        SP_HPivRnd_18_Xe.trans.X := g_H_sideplateDIST + NOZZLE_RADIUS;
        SP_HPivRnd_18_Xs.trans.X := g_H_sideplateDIST + NOZZLE_RADIUS + 50 ;
        SP_gPivRnd_18_Xe.trans.X := ( g_H_sideplateDIST + NOZZLE_RADIUS ) * (-1);
        SP_gPivRnd_18_Xs.trans.X := ( g_H_sideplateDIST + NOZZLE_RADIUS + 50) * (-1);

        SP_HPivRnd_18_Xe.trans.y := yy_SRCH_Target ;
        SP_HPivRnd_18_Xs.trans.y := yy_SRCH_Target;
        SP_gPivRnd_18_Xe.trans.y := yy_SRCH_Target ;
        SP_gPivRnd_18_Xs.trans.y := yy_SRCH_Target;

        SP_HPivRnd_18_Xe.trans.z := zz_SRCH_Target * (-1) ;
        SP_HPivRnd_18_Xs.trans.z := zz_SRCH_Target * (-1) ;
        SP_gPivRnd_18_Xe.trans.z := zz_SRCH_Target * (-1) ;
        SP_gPivRnd_18_Xs.trans.z := zz_SRCH_Target * (-1) ;

 !!!!!!!!!!!!!!!!!!!!!!!!!!!!!!!!!!!!!!!!!!!!!!!!!!!!!!!!!!!!!!!!!!!!!!!!!!!!!

        SP_hPivCam_18_Xe.trans.X := g_H_sideplateDIST - NOZZLE_RADIUS;
        SP_hPivCam_18_Xs.trans.X := g_H_sideplateDIST - NOZZLE_RADIUS - 50 ;
        SP_gPivCam_18_Xe.trans.X := (g_H_sideplateDIST -  NOZZLE_RADIUS) *(-1);
        SP_gPivCam_18_Xs.trans.X := (g_H_sideplateDIST - NOZZLE_RADIUS - 50) * (-1) ;

        SP_hPivCam_18_Xe.trans.y := yy_SRCH_Target ;
        SP_hPivCam_18_Xs.trans.y := yy_SRCH_Target;
        SP_gPivCam_18_Xe.trans.y := yy_SRCH_Target ;
        SP_gPivCam_18_Xs.trans.y := yy_SRCH_Target;

        SP_hPivCam_18_Xe.trans.z := zz_SRCH_Target * (-1) ;
        SP_hPivCam_18_Xs.trans.z := zz_SRCH_Target * (-1) ;
        SP_gPivCam_18_Xe.trans.z := zz_SRCH_Target * (-1) ;
        SP_gPivCam_18_Xs.trans.z := zz_SRCH_Target * (-1) ;

        SP_HPivRnd_PJ_Xe.trans.X := g_H_sideplateDIST - NOZZLE_RADIUS - SIDEPLATE;
        SP_HPivRnd_PJ_Xs.trans.X := g_H_sideplateDIST - NOZZLE_RADIUS - SIDEPLATE - 50;
        SP_gPivRnd_PJ_Xe.trans.X := (g_H_sideplateDIST - NOZZLE_RADIUS - SIDEPLATE) *(-1);
        SP_gPivRnd_PJ_Xs.trans.X := (g_H_sideplateDIST - NOZZLE_RADIUS - SIDEPLATE - 50) * (-1);

        SP_HPivRnd_PJ_Xe.trans.y := yy_SRCH_Target;
        SP_HPivRnd_PJ_Xs.trans.y := yy_SRCH_Target;
        SP_gPivRnd_PJ_Xe.trans.y := yy_SRCH_Target;
        SP_gPivRnd_PJ_Xs.trans.y := yy_SRCH_Target;

        SP_HPivRnd_PJ_Xe.trans.z := zz_SRCH_Target * (-1);
        SP_HPivRnd_PJ_Xs.trans.z := zz_SRCH_Target * (-1);
        SP_gPivRnd_PJ_Xe.trans.z := zz_SRCH_Target * (-1) ;
        SP_gPivRnd_PJ_Xs.trans.z := zz_SRCH_Target * (-1) ;

 !!!!!!!!!!!!!!!!!!!!!!!!!!!!!!!!!!!!!!!!!!!!!!!!!!!!!!!!!!!!!!!!!!!!!!!!!!!!!

        SP_hPivCam_PJ_Xe.trans.X := g_H_sideplateDIST + SIDEPLATE + NOZZLE_RADIUS;
        SP_hPivCam_PJ_Xs.trans.X := g_H_sideplateDIST + SIDEPLATE + NOZZLE_RADIUS + 50;
        SP_gPivCam_PJ_Xe.trans.X := (g_H_sideplateDIST + SIDEPLATE + NOZZLE_RADIUS) * (-1);
        SP_gPivCam_PJ_Xs.trans.X := (g_H_sideplateDIST + SIDEPLATE + NOZZLE_RADIUS + 50) * (-1);

        SP_hPivCam_PJ_Xe.trans.y := yy_SRCH_Target;
        SP_hPivCam_PJ_Xs.trans.y := yy_SRCH_Target;
        SP_gPivCam_PJ_Xe.trans.y := yy_SRCH_Target;
        SP_gPivCam_PJ_Xs.trans.y := yy_SRCH_Target;

        SP_hPivCam_PJ_Xe.trans.z := zz_SRCH_Target * (-1);
        SP_hPivCam_PJ_Xs.trans.z := zz_SRCH_Target * (-1);
        SP_gPivCam_PJ_Xe.trans.z := zz_SRCH_Target * (-1);
        SP_gPivCam_PJ_Xs.trans.z := zz_SRCH_Target * (-1);

!!!!!!!!!!!!!!!!!!!!!!!!!!!!!!!!!!!!!!!!!!!!!!!!!!!!!!!!!!!!!!!!!!!!!!!!!!!!!!!!!!!!!!!!!!!!!!!!!!!!!!
        SP_GRnd_Side_XE.TRANS.X := (g_H_sideplateDIST + NOZZLE_RADIUS) *(-1);
        SP_GRnd_Side_XS.TRANS.X := (g_H_sideplateDIST + NOZZLE_RADIUS + 50) *(-1);
        SP_GRnd_Side_XE.trans.y := yy_SRCH_Target;
        SP_GRnd_Side_XS.trans.y := yy_SRCH_Target;
        SP_GRnd_Side_XE.trans.z := zz_SRCH_Target * (-1);
        SP_GRnd_Side_XS.trans.z := zz_SRCH_Target * (-1);
        SP_GRnd_Side_XS.extax.eax_b := 0;
        SP_GRnd_Side_XS.extax.eax_c := 90;
        SP_GRnd_Side_XE.extax := SP_GRnd_Side_XS.extax;

        SP_HRnd_Side_XE.TRANS.X := (g_H_sideplateDIST + NOZZLE_RADIUS) ;
        SP_HRnd_Side_XS.TRANS.X := (g_H_sideplateDIST + NOZZLE_RADIUS + 50) ;
        SP_HRnd_Side_XE.trans.y := yy_SRCH_Target;
        SP_HRnd_Side_XS.trans.y := yy_SRCH_Target;
        SP_HRnd_Side_XE.trans.z := zz_SRCH_Target * (-1);
        SP_HRnd_Side_XS.trans.z := zz_SRCH_Target * (-1);
        SP_HRnd_Side_XS.extax.eax_b := 0;
        SP_HRnd_Side_XS.extax.eax_c := -90;
        SP_HRnd_Side_XE.extax := SP_HRnd_Side_XS.extax;

        SP_GCam_Side_XE.TRANS.X := (g_H_sideplateDIST + NOZZLE_RADIUS + SIDEPLATE) *(-1);
        SP_GCam_Side_XS.TRANS.X := (g_H_sideplateDIST + NOZZLE_RADIUS + SIDEPLATE + 50) *(-1);
        SP_GCam_Side_XE.trans.y := yy_SRCH_Target;
        SP_GCam_Side_XS.trans.y := yy_SRCH_Target;
        SP_GCam_Side_XE.trans.z := zz_SRCH_Target * (-1);
        SP_GCam_Side_XS.trans.z := zz_SRCH_Target * (-1);
        SP_GCam_Side_XE.extax := g29.extax;
        SP_GCam_Side_XS.extax := g29.extax;

        SP_HCam_Side_XE.TRANS.X := (g_H_sideplateDIST + NOZZLE_RADIUS + SIDEPLATE) ;
        SP_HCam_Side_XS.TRANS.X := (g_H_sideplateDIST + NOZZLE_RADIUS + SIDEPLATE + 50) ;
        SP_HCam_Side_XE.trans.y := yy_SRCH_Target;
        SP_HCam_Side_XS.trans.y := yy_SRCH_Target;
        SP_HCam_Side_XE.trans.z := zz_SRCH_Target * (-1);
        SP_HCam_Side_XS.trans.z := zz_SRCH_Target * (-1);
        SP_HCam_Side_XE.extax := H29.extax;
        SP_HCam_Side_XS.extax := H29.extax;

        SP_Piv0ut_GXe.trans.X := (g_H_sideplateDIST - NOZZLE_RADIUS) * (-1) ;
        SP_Piv0ut_GXs.trans.X := (g_H_sideplateDIST - NOZZLE_RADIUS - 50) * (-1) ;
        SP_Piv0ut_HXe.trans.X := (g_H_sideplateDIST - NOZZLE_RADIUS)  ;
        SP_Piv0ut_HXs.trans.X := (g_H_sideplateDIST - NOZZLE_RADIUS - 50)  ;

        SP_Piv0ut_GXe.trans.y := yy_SRCH_Target ;
        SP_Piv0ut_GXs.trans.y := yy_SRCH_Target ;
        SP_Piv0ut_GXe.trans.z := zz_SRCH_Target * (-1);
        SP_Piv0ut_GXs.trans.z := zz_SRCH_Target * (-1);

        SP_Piv0ut_HXe.trans.y := yy_SRCH_Target ;
        SP_Piv0ut_HXs.trans.y := yy_SRCH_Target ;
        SP_Piv0ut_HXe.trans.z := zz_SRCH_Target * (-1);
        SP_Piv0ut_HXs.trans.z := zz_SRCH_Target * (-1);

        IF pivCAM = TRUE THEN
            XH0E.TRANS.X := (g_H_sideplateDIST + SIDEPLATE + NOZZLE_RADIUS);
            XH19E.TRANS.X := (g_H_sideplateDIST + SIDEPLATE + NOZZLE_RADIUS);
            XH29E.TRANS.X := (g_H_sideplateDIST + SIDEPLATE + NOZZLE_RADIUS);

            XG0E.TRANS.X := (g_H_sideplateDIST + SIDEPLATE + NOZZLE_RADIUS) * (-1);
            XG19E.TRANS.X := (g_H_sideplateDIST + SIDEPLATE + NOZZLE_RADIUS) * (-1);
            XG29E.TRANS.X :=  (g_H_sideplateDIST + SIDEPLATE + NOZZLE_RADIUS) * (-1);

            XL49E.TRANS.X := (g_H_sideplateDIST + SIDEPLATE + NOZZLE_RADIUS);
            XM49E.TRANS.X := (g_H_sideplateDIST - NOZZLE_RADIUS) * (-1) ;
        ELSEIF PIVCAM = FALSE THEN
            XH0E.TRANS.X := (g_H_sideplateDIST + NOZZLE_RADIUS);
            XH19E.TRANS.X := (g_H_sideplateDIST  + NOZZLE_RADIUS);
            XH29E.TRANS.X := (g_H_sideplateDIST  + NOZZLE_RADIUS);

            XG0E.TRANS.X := (g_H_sideplateDIST + NOZZLE_RADIUS) * (-1);
            XG19E.TRANS.X := (g_H_sideplateDIST + NOZZLE_RADIUS) * (-1);
            XG29E.TRANS.X :=  (g_H_sideplateDIST + NOZZLE_RADIUS) * (-1);

            XL49E.TRANS.X := (g_H_sideplateDIST  + NOZZLE_RADIUS);
            XM49E.TRANS.X := (g_H_sideplateDIST - SIDEPLATE - NOZZLE_RADIUS) * (-1) ;
        ENDIF
        WAITTIME\INPOS,.2;
    ENDPROC

    PROC Piv_side_Welds(string RND_OR_NOT)

	 IF PIVOT_USED = 6089330 OR PIVOT_USED = 6802774 OR PIVOT_USED = 6870131 OR PIVOT_USED = 6845931 THEN
     !!  THIS IS FOR A 42H, 33H AND 24H
	    pivCAM := FALSE;

 	ELSEIF PIVOT_USED =  674961 OR PIVOT_USED = 350404 OR PIVOT_USED = 6099018 THEN
     !!  THIS IS FOR 77F THRU 120F AND 18H !
        pivCAM := TRUE;

	ELSE STOP;

	ENDIF

	WAITTIME\INPOS,.1;

	IF RND_OR_NOT = "G" AND pivCAM = TRUE THEN
		GOTO G_CAM_SIDE_WELDS;

	ELSEIF RND_OR_NOT = "G" AND pivCAM = FALSE THEN
		GOTO G_RND_SIDE_WELDS;

	ELSEIF RND_OR_NOT = "H" AND pivCAM = TRUE THEN
		GOTO H_CAM_SIDE_WELDS;

	ELSEIF RND_OR_NOT = "H" AND pivCAM = FALSE THEN
		GOTO H_RND_SIDE_WELDS;

    ELSE STOP;

	ENDIF
 G_RND_SIDE_WELDS:
        ! This is executed only if the Pivot is ROUND in Shape
       	ActUnit STN1;
        BEGIN_TEST_WELD_Grnd_OUTSIDE:
        MoveJ Offs(SP_GRnd_Side_XS, -300, 0, 0), V500, z10, tWeldGun\WObj:=wobj_PivCam;
        MoveL Offs(SP_GRnd_Side_XS, -50, 0, 0), V500, z5, tWeldGun\WObj:=wobj_PivCam;
        Search_1D SR_GSide_X\SearchStop:=gX_SideFOUND, SP_GRnd_Side_XS, SP_GRnd_Side_XE, v50, tWeldGun\WObj:=wobj_PivCam\SchSpeed:=10;
        MoveL Offs(SP_GRnd_Side_XS, -100, 0, 0), V500, z5, tWeldGun\WObj:=wobj_PivCam;
        MoveJ Offs(SP_GRnd_Side_YS, -120, 100, 0), V500, z10, tWeldGun\WObj:=wobjHsideplate;
        PivG_SideYZ_XSET_18_R1 gX_SideFOUND ;
        MoveL offs(SP_GRnd_Side_YS,-120,75,0), V500, z5, tWeldGun\WObj:=wobjHsideplate;
        MoveL offs(SP_GRnd_Side_YS,0,75,0), V500, z5, tWeldGun\WObj:=wobjHsideplate;
        Search_1D SR_GSide_Y\SearchStop:=gY_SideFOUND, SP_GRnd_Side_YS, SP_GRnd_Side_YE, v300, tWeldGun\WObj:=wobjHsideplate\SchSpeed:=10;
  		MoveL gY_SideFOUND, V500, z1, tWeldGun\WObj:=wobjHsideplate;
        WaitTime\InPos, 1;
        PivFOUND_Y := CRobT(\Tool:=tWeldgun\WObj:=obSTN1);
        WaitTime\InPos, 1;
        MoveL offs(SP_GRnd_Side_YS,0,50,0), V500, z5, tWeldGun\WObj:=wobjHsideplate;
        MoveL offs(SP_GRnd_Side_YS,-150,100,0), V500, z10, tWeldGun\WObj:=wobjHsideplate;
        MoveJ offs(SP_GRnd_Side_ZS,-150,0,100), V500, z10, tWeldGun\WObj:=wobjHsideplate;
        MoveL offs(SP_GRnd_Side_ZS,0,0,50), v400, z10, tWeldGun\WObj:=wobjHsideplate;
        Search_1D SR_GSide_Z\SearchStop:=gZ_SideFOUND, SP_GRnd_Side_ZS, SP_GRnd_Side_ZE, v300, tWeldGun\WObj:=wobjHsideplate\SchSpeed:=10;
  		MoveL gZ_SideFOUND, V500, z1, tWeldGun\WObj:=wobjHsideplate;
        WaitTime\InPos, 1;
        PivFOUND_Z := CRobT(\Tool:=tWeldgun\WObj:=obSTN1);
        WaitTime\InPos, 1;
        MoveL offs(SP_GRnd_Side_ZS,0,0,75), V500, z5, tWeldGun\WObj:=wobjHsideplate;
        PivWobj_Translation_Locator wobj_PivCam, PivFOUND_Y, PivFOUND_Z, WPIVOTANGLE;
        WaitTime\inpos, 1;
        MoveJ offs(SP_GRnd_Side_ZS,-300,0,75), V500, z10, tWeldGun\WObj:=wobjHsideplate;
        MoveJ Offs(GRnd_SidePIV_S,-300,200,0), V500, z10, tWeldGun\WObj:=wobj_PivCam;
        Search_1D SRpivotYhelperGsideRound,Offs(SPpivotYhelperGsideRoundE,0,30,0), SPpivotYhelperGsideRoundE, v100, tWeldGun\WObj:=wobj_PivCam\SchSpeed:=10;
        MoveJ Offs(GRnd_SidePIV_S,-300,200,0), V500, z10, tWeldGun\WObj:=wobj_PivCam;
        MoveJ offs(GRnd_SidePIV_S,-300,0,0), V500, z10, tWeldGun\WObj:=wobj_PivCam;
        PDispSet SRpivotYhelperGsideRound;
        ArcLStart GRnd_SidePIV_S, v100, smGH40A, wdGH40B\Weave:=wvGH40B, z1, tWeldGun\WObj:=wobj_PivCam;
		ArcL Offs(GRnd_SidePIV_S,0,0,5), v100, smGH40A, wdGH40B\Weave:=wvGH40B, z1, tWeldGun\WObj:=wobj_PivCam;
		WaitTime\InPos, 0.5;
		ArcL GRnd_SidePIV_Sm, v100, smGH40A, wdGH40B\Weave:=wvGH40B, z1, tWeldGun\WObj:=wobj_PivCam;
		ArcL GRnd_SidePIV_M, v100, smGH40A, wdGH40A\Weave:=wvGH40A, z1, tWeldGun\WObj:=wobj_PivCam;
		ArcL GRnd_SidePIV_Em, v100, smGH40A, wdGH40C\Weave:=wv0, z1, tWeldGun\WObj:=wobj_PivCam;
		ArcLEnd GRnd_SidePIV_E, v100, smGH40A, wdGH40C\Weave:=wv0, z1, tWeldGun\WObj:=wobj_PivCam;
        PDispOff;
        MoveL offs(GRnd_SidePIV_E,-50,0,0), V500, z10, tWeldGun\WObj:=wobj_PivCam;
        MoveJ offs(GRnd_SidePIV_E,-600,0,0), V500, z10, tWeldGun\WObj:=wobj_PivCam;
        WELDED_GRND_OUTSIDE:
        GOTO GLUED_THE_PIV_SIDES;
G_CAM_SIDE_WELDS:
        ! This is executed only if the Pivot is CAM in Shape
       	ActUnit STN1;
        BEGIN_TEST_WELD_GCam_OUTSIDE:
        PivG_SideYZ_XSET_18_R1 Gx_weld_piv;
        WAITTIME\INPOS, 1;
        firstYthentheZ:
        MoveJ Offs(SP_GCam_Side_YS, -175, 100, 0), V500, z10, tWeldGun\WObj:=wobjHsideplate;
        MoveL offs(SP_GCam_Side_YS,0,75,0), V500, z5, tWeldGun\WObj:=wobjHsideplate;
        Search_1D SR_GSide_Y\SearchStop:=gY_SideFOUND, SP_GCam_Side_YS, SP_GCam_Side_YE, v300, tWeldGun\WObj:=wobjHsideplate\SchSpeed:=10;
  		MoveL gY_SideFOUND, V500, z1, tWeldGun\WObj:=wobjHsideplate;
        WaitTime\InPos, 1;
        PivFOUND_Y := CRobT(\Tool:=tWeldgun\WObj:=obSTN1);
        WaitTime\InPos, 1;
        MoveL offs(SP_GCam_Side_YS,0,50,0), V500, z5, tWeldGun\WObj:=wobjHsideplate;
        MoveL offs(SP_GCam_Side_YS,-150,100,0), V500, z10, tWeldGun\WObj:=wobjHsideplate;
        nowtheZ:
        MoveJ offs(SP_GCam_Side_ZS,-150,0,100), V500, z10, tWeldGun\WObj:=wobjHsideplate;
        MoveL offs(SP_GCam_Side_ZS,0,0,50), v400, z10, tWeldGun\WObj:=wobjHsideplate;
        Search_1D SR_GSide_Z\SearchStop:=gZ_SideFOUND, SP_GCam_Side_ZS, SP_GCam_Side_ZE, v300, tWeldGun\WObj:=wobjHsideplate\SchSpeed:=10;
  		MoveL gZ_SideFOUND, V500, z1, tWeldGun\WObj:=wobjHsideplate;
        WaitTime\InPos, 1;
        PivFOUND_Z := CRobT(\Tool:=tWeldgun\WObj:=obSTN1);
        WaitTime\InPos, 1;
        MoveL offs(SP_GCam_Side_ZS,0,0,75), V500, z5, tWeldGun\WObj:=wobjHsideplate;
        PivWobj_Translation_Locator wobj_PivCam, PivFOUND_Y, PivFOUND_Z, WPIVOTANGLE;
        WaitTime\inpos, 1;
        MoveL offs(SP_GCam_Side_ZS,-300,0,75), V500, z10, tWeldGun\WObj:=wobjHsideplate;
        MoveJ RelTooL(GCam_SidePIV_S,0,0,-350), V500, z10, tWeldGun\WObj:=wobj_PivCam;
        WELDED_GCAM_OUTSIDE:
        GOTO GLUED_THE_PIV_SIDES;
 H_CAM_SIDE_WELDS:
            ! This is executed only if the Pivot is CAM in Shape
       	ActUnit STN1;
        BEGIN_TEST_WELD_HCam_OUTSIDE:
        PivH_SideYZ_XSET_18_R1 hx_weld_piv;
        MoveJ Offs(SP_HCam_Side_YS, 200, 100, 0), V500, z10, tWeldGun\WObj:=wobjHsideplate;
        MoveL offs(SP_HCam_Side_YS,0,75,0), V500, z5, tWeldGun\WObj:=wobjHsideplate;
        Search_1D SR_HSide_Y\SearchStop:=hY_SideFOUND, SP_HCam_Side_YS, SP_HCam_Side_YE, v300, tWeldGun\WObj:=wobjHsideplate\SchSpeed:=10;
  		MoveL hY_SideFOUND, V500, z1, tWeldGun\WObj:=wobjHsideplate;
        WaitTime\InPos, 1;
        PivFOUND_Y := CRobT(\Tool:=tWeldgun\WObj:=obSTN1);
        WaitTime\InPos, 1;
        MoveL offs(SP_HCam_Side_YS,0,50,0), V500, z5, tWeldGun\WObj:=wobjHsideplate;
        MoveL offs(SP_HCam_Side_YS,150,100,0), V500, z10, tWeldGun\WObj:=wobjHsideplate;
        MoveJ offs(SP_HCam_Side_ZS,150,0,100), V500, z10, tWeldGun\WObj:=wobjHsideplate;
        MoveL offs(SP_HCam_Side_ZS,0,0,50), v400, z10, tWeldGun\WObj:=wobjHsideplate;
        Search_1D SR_HSide_Z\SearchStop:=hZ_SideFOUND, SP_HCam_Side_ZS, SP_HCam_Side_ZE, v300, tWeldGun\WObj:=wobjHsideplate\SchSpeed:=10;
  		MoveL hZ_SideFOUND, V500, z1, tWeldGun\WObj:=wobjHsideplate;
        WaitTime\InPos, 1;
        PivFOUND_Z := CRobT(\Tool:=tWeldgun\WObj:=obSTN1);
        WaitTime\InPos, 1;
        MoveL offs(SP_HCam_Side_ZS,0,0,75), V500, z5, tWeldGun\WObj:=wobjHsideplate;
        PivWobj_Translation_Locator wobj_PivCam, PivFOUND_Y, PivFOUND_Z, WPIVOTANGLE;
        WaitTime\inpos, 1;
        MoveL offs(SP_HCam_Side_ZS,0,-300,0), V500, z10, tWeldGun\WObj:=wobjHsideplate;
        MoveJ reltool(HCam_SidePIV_S,0,0,-300), V500, z10, tWeldGun\WObj:=wobj_PivCam;
        WELDED_HCAM_OUTSIDE:
        GOTO GLUED_THE_PIV_SIDES;
 H_RND_SIDE_WELDS:
        ! This is executed only if the Pivot is ROUND in Shape
       	ActUnit STN1;
        BEGIN_TEST_WELD_HRnd_OUTSIDE:
        MoveJ Offs(SP_HRnd_Side_XS, 300, 0, 0), V500, z10, tWeldGun\WObj:=wobj_PivCam;
        MoveL Offs(SP_HRnd_Side_XS, 50, 0, 0), V500, z5, tWeldGun\WObj:=wobj_PivCam;
        Search_1D SR_HSide_X\SearchStop:=hX_SideFOUND, SP_HRnd_Side_XS, SP_HRnd_Side_XE, v50, tWeldGun\WObj:=wobj_PivCam\SchSpeed:=10;
        MoveL Offs(SP_HRnd_Side_XS, 100, 0, 0), V500, z5, tWeldGun\WObj:=wobj_PivCam;
        PivH_SideYZ_XSET_18_R1 hX_SideFOUND;
        MoveJ Offs(SP_HRnd_Side_YS, 100, 100, 0), V500, z10, tWeldGun\WObj:=wobjHsideplate;
        MoveL offs(SP_HRnd_Side_YS,0,75,0), V500, z5, tWeldGun\WObj:=wobjHsideplate;
        Search_1D SR_HSide_Y\SearchStop:=hY_SideFOUND, SP_HRnd_Side_YS, SP_HRnd_Side_YE, v300, tWeldGun\WObj:=wobjHsideplate\SchSpeed:=10;
  		MoveL hY_SideFOUND, V500, z1, tWeldGun\WObj:=wobjHsideplate;
        WaitTime\InPos, 1;
        PivFOUND_Y := CRobT(\Tool:=tWeldgun\WObj:=obSTN1);
        WaitTime\InPos, 1;
        MoveL offs(SP_HRnd_Side_YS,0,50,0), V500, z5, tWeldGun\WObj:=wobjHsideplate;
        MoveL offs(SP_HRnd_Side_YS,150,100,0), V500, z10, tWeldGun\WObj:=wobjHsideplate;
        MoveJ offs(SP_HRnd_Side_ZS,150,0,100), V500, z10, tWeldGun\WObj:=wobjHsideplate;
        MoveL offs(SP_HRnd_Side_ZS,0,0,50), v400, z10, tWeldGun\WObj:=wobjHsideplate;
        Search_1D SR_HSide_Z\SearchStop:=hZ_SideFOUND, SP_HRnd_Side_ZS, SP_HRnd_Side_ZE, v300, tWeldGun\WObj:=wobjHsideplate\SchSpeed:=10;
  		MoveL hZ_SideFOUND, V500, z1, tWeldGun\WObj:=wobjHsideplate;
        WaitTime\InPos, 1;
        PivFOUND_Z := CRobT(\Tool:=tWeldgun\WObj:=obSTN1);
        WaitTime\InPos, 1;
        MoveL offs(SP_HRnd_Side_ZS,0,0,75), V500, z5, tWeldGun\WObj:=wobjHsideplate;
        PivWobj_Translation_Locator wobj_PivCam, PivFOUND_Y, PivFOUND_Z, WPIVOTANGLE;
        WaitTime\inpos, 1;
        MoveL offs(SP_HRnd_Side_ZS,300,0,75), V500, z10, tWeldGun\WObj:=wobjHsideplate;
        MoveJ Offs(HRnd_SidePIV_S,300,200,0), V500, z10, tWeldGun\WObj:=wobj_PivCam;
        Search_1D SRpivotYhelperHsideRound,Offs(SPpivotYhelperHsideRoundE,0,30,0), SPpivotYhelperHsideRoundE, v100, tWeldGun\WObj:=wobj_PivCam\SchSpeed:=10;
        MoveJ Offs(HRnd_SidePIV_S,300,200,0), V500, z10, tWeldGun\WObj:=wobj_PivCam;
        MoveJ offs(HRnd_SidePIV_S,300,0,0), V500, z10, tWeldGun\WObj:=wobj_PivCam;
        MoveJ offs(HRnd_SidePIV_S,300,0,0), V500, z10, tWeldGun\WObj:=wobj_PivCam;
        PDispSet SRpivotYhelperHsideRound;
 		ArcLStart HRnd_SidePIV_S, v100, smGH40A, wdGH40B\Weave:=wvGH40B, z1, tWeldGun\WObj:=wobj_PivCam;
		ArcL Offs(HRnd_SidePIV_S,0,0,5), v100, smGH40A, wdGH40B\Weave:=wvGH40B, z1, tWeldGun\WObj:=wobj_PivCam;
		WaitTime\InPos, 0.5;
		ArcL HRnd_SidePIV_Sm, v100, smGH40A, wdGH40B\Weave:=wvGH40B, z1, tWeldGun\WObj:=wobj_PivCam;
		ArcL HRnd_SidePIV_M, v100, smGH40A, wdGH40A\Weave:=wvGH40A, z1, tWeldGun\WObj:=wobj_PivCam;
		ArcL HRnd_SidePIV_Em, v100, smGH40A, wdGH40C\Weave:=wv0, z1, tWeldGun\WObj:=wobj_PivCam;
		ArcLEnd HRnd_SidePIV_E, v100, smGH40A, wdGH40C\Weave:=wv0, z1, tWeldGun\WObj:=wobj_PivCam;
        PDispOff;
        MoveL offs(HRnd_SidePIV_E,50,0,0), V500, z10, tWeldGun\WObj:=wobj_PivCam;
        MoveJ offs(HRnd_SidePIV_E,600,0,0), V500, z10, tWeldGun\WObj:=wobj_PivCam;
        WELDED_HRnd_OUTSIDE:
        GOTO GLUED_THE_PIV_SIDES;
      GLUED_THE_PIV_SIDES:
    ENDPROC

        PROC Piv0ut2Fwrap_X18_R1()

                SP_Piv0ut_Ye.trans.X := (hX_FOUND.TRANS.X) + (NOZZLE_RADIUS * 1.5)  ;
                SP_Piv0ut_Ys.trans.X := (hX_FOUND.TRANS.X) + (NOZZLE_RADIUS * 1.5)  ;
                SP_Piv0ut_Ye.trans.y := NOZZLE_RADIUS ;
                SP_Piv0ut_Ys.trans.y := NOZZLE_RADIUS + 55;

                SP_Piv0ut_Ye.trans.z := wobjHpivot.oframe.trans.Z - 164 ;
                SP_Piv0ut_Ys.trans.z := wobjHpivot.oframe.trans.Z - 164 ;
                SP_Piv0ut_Ze.trans.X := (hX_FOUND.TRANS.X) + (NOZZLE_RADIUS*1.5) ;
                SP_Piv0ut_Zs.trans.X := (hX_FOUND.TRANS.X) + (NOZZLE_RADIUS*1.5) ;

                SP_Piv0ut_Ze.trans.Y := 36;
                SP_Piv0ut_Zs.trans.Y := 36;
                SP_Piv0ut_Ze.trans.z := (wobjHpivot.oframe.trans.Z)  - hfixconst + nozzle_radius ;
                SP_Piv0ut_Zs.trans.z := (wobjHpivot.oframe.trans.Z - HFIXCONST + NOZZLE_RADIUS + 50) ;
            over_it:
    ENDPROC

    PROC Weld_Piv0ut_2FWrap()
       ActUnit STN1;
       PDispOff;
       PDispOff;
       MoveJ pjthomeSTA1zero, vCellSpeed, fine, tWeldGun\WObj:=wobj0;
       MoveJ RelTool(SP_Piv0ut_GXs,0,0,-650), V500, z20, tWeldGun\WObj:=wobj_PivCam;
       MoveL RelTool(SP_Piv0ut_GXs,0,0,-150), V500, z5, tWeldGun\WObj:=wobj_PivCam;
       PDispOff;
       MoveL SP_Piv0ut_GXs, V500, z1, tWeldGun\WObj:=wobj_PivCam;
       Search_1D SR_Gx\SearchStop:=gX_FOUND, SP_Piv0ut_GXs, SP_Piv0ut_GXe, v300, tWeldGun\WObj:=wobj_PivCam\SchSpeed:=10;
       MoveL RelTool(SP_Piv0ut_GXs,0,0,-50), V500, z5, tWeldGun\WObj:=wobj_PivCam;
       MoveL RelTool(SP_Piv0ut_HXs,0,0,-50), V500, z5, tWeldGun\WObj:=wobj_PivCam;
       Search_1D SR_Hx\SearchStop:=hX_FOUND, SP_Piv0ut_HXs, SP_Piv0ut_HXe, v300, tWeldGun\WObj:=wobj_PivCam\SchSpeed:=10;
       MoveL RelTool(SP_Piv0ut_HXs,0,0,-150), V500, z5, tWeldGun\WObj:=wobj_PivCam;
       Piv0ut2Fwrap_X18_R1;
       MoveJ Offs(SP_Piv0ut_Zs,0,-250,0), V500, z5, tWeldGun\WObj:=wobjHsideplate;
       MoveJ Offs(SP_Piv0ut_Zs,250,-250,0), V500, z5, tWeldGun\WObj:=wobjHsideplate;
       MoveJ Offs(SP_Piv0ut_Ys,250,0,50), V500, z5, tWeldGun\WObj:=wobjHsideplate;
       Search_1D SR_Piv_Y\SearchStop:=PivFOUND_Y, SP_Piv0ut_Ys, SP_Piv0ut_Ye, v300, tWeldGun\WObj:=wobjHsideplate\PrePDisp:=SR_Hx\SchSpeed:=10;
  	   MoveL PivFOUND_Y, V500, z1, tWeldGun\WObj:=wobjHsideplate;
       PDispOff;
       WaitTime\InPos, 1;
       PivFOUND_Y := CRobT(\Tool:=tWeldGun\WObj:=obSTN1);
       WaitTime\InPos, 1;
       MoveL Offs(SP_Piv0ut_Ys,0,50,0), V500, z5, tWeldGun\WObj:=wobjHsideplate;
       MoveL OFFS(SP_Piv0ut_Ys,250,0,50), V500, z5, tWeldGun\WObj:=wobjHsideplate;
       MoveJ OFFS(SP_Piv0ut_Zs,200,0,150), V500, z5, tWeldGun\WObj:=wobjHsideplate;
       MoveL OFFS(SP_Piv0ut_Zs,200,0,50), V500, z5, tWeldGun\WObj:=wobjHsideplate;
       Search_1D SR_Piv_Z\SearchStop:=PivFOUND_z, SP_Piv0ut_Zs, SP_Piv0ut_Ze, v300, tWeldGun\WObj:=wobjHsideplate\PrePDisp:=SR_Piv_Y\SchSpeed:=10;
  	   MoveL PivFOUND_z, V500, z1, tWeldGun\WObj:=wobjHsideplate;
       PDispOff;
       WaitTime\InPos, 1;
       PivFOUND_z := CRobT(\Tool:=tWeldGun\WObj:=obSTN1);
       WaitTime\InPos, 1;
       MoveL OFFS(SP_Piv0ut_Zs,0,-50,100), V500, z5, tWeldGun\WObj:=wobjHsideplate;
       MoveL OFFS(SP_Piv0ut_Zs,200,50,0), V500, z5, tWeldGun\WObj:=wobjHsideplate;
        PivWobj_Translation_Locator wobj_PivCam, PivFOUND_Y, PivFOUND_Z, WPIVOTANGLE;
        WaitTime\InPos, 1;
       !MoveL OFFS(SP_Piv0ut_Ys,200,-300,0), V500, z5, tWeldGun\WObj:=wobjHsideplate;
       MoveJ OFFS(SP_Piv0ut_Zs,200,-300,0), V500, z5, tWeldGun\WObj:=wobjHsideplate;
       MoveJ OFFS(SP_Piv0ut_Zs,-100,-300,0), V500, z5, tWeldGun\WObj:=wobjHsideplate;
       MoveJ OFFS(OSPiv2Fwrap_G1,100,-200,0), V500, z5, tWeldGun\WObj:=wobj_PivCam;
       !Y and Z SEARCH FOR DISP...03-19-18
       Search_1D SR_YPIVadj,Offs(SP_YPIVadj_e,0,-30,0), SP_YPIVadj_e, v300, tWeldGun\WObj:=wobj_PivCam\SchSpeed:=10;
       MoveJ OFFS(OSPiv2Fwrap_G1,100,-200,0), V500, z5, tWeldGun\WObj:=wobj_PivCam;
       Search_1D\Wire, SR_ZPIVadj, Offs(SP_ZPIVadj_e,0,-10,-30), SP_ZPIVadj_e, v300, tWeldGun\WObj:=wobj_PivCam\SchSpeed:=10;
       MoveJ OFFS(OSPiv2Fwrap_G1,100,-200,0), V500, z5, tWeldGun\WObj:=wobj_PivCam;
		SR_Gx.trans.y := SR_YPIVadj.trans.y;
		SR_Gx.trans.z := SR_ZPIVadj.trans.z;
		SR_Hx.trans.y := SR_YPIVadj.trans.y;
		SR_Hx.trans.z := SR_ZPIVadj.trans.z;
        WaitTime\InPos, 1;
        TPErase;
        TPErase;
       PDispSet SR_Gx;
	   ArcLStart OSPiv2Fwrap_G3, v100, smJKnofill, wdJKroot\Weave:=wvJKroot, z1, tWeldGun\WObj:=wobj_PivCam;
       PDispSet SR_Hx;
       ArcLEnd OSPiv2Fwrap_H3, v100, smJKnofill, wdJKroot\Weave:=wvJKroot, z1, tWeldGun\WObj:=wobj_PivCam;
       MoveL Offs(OSPiv2Fwrap_H3,0,-35,0), v100, z1, tWeldGun\WObj:=wobj_PivCam;
       PDispOff;
	   MoveL Offs(OSPiv2Fwrap_G1,35,-35,0), v300, z1, tWeldGun\WObj:=wobj_PivCam;
       PDispSet SR_Gx;
       ArcLStart OSPiv2Fwrap_G1, v100, smJK1, wdJK1\Weave:=wv0, z1, tWeldGun\WObj:=wobj_PivCam\Track:=track0;
	   ArcL OSPiv2Fwrap_G2, v100, smJK, wdJK1\Weave:=wv0, z1, tWeldGun\WObj:=wobj_PivCam\Track:=track0;
	   ArcL OSPiv2Fwrap_G3, v100, smJK, wdJK1\Weave:=wvJK, z1, tWeldGun\WObj:=wobj_PivCam\Track:=track0;
	   ArcLEnd OSPiv2Fwrap_G4, v100, smJKnofill, wdJK\Weave:=wvJK, z1, tWeldGun\WObj:=wobj_PivCam\Track:=trLM10hiteonly;
	   PDispOff;
       MoveL Offs(OSPiv2Fwrap_G4,0,-35,0), v100, z1, tWeldGun\WObj:=wobj_PivCam;
	   MoveL Offs(OSPiv2Fwrap_H1,-35,-35,0), v100, z1, tWeldGun\WObj:=wobj_PivCam;
       PDispSet SR_Hx;
       ArcLStart OSPiv2Fwrap_H1, v100, smJK1, wdJK1\Weave:=wv0, z1, tWeldGun\WObj:=wobj_PivCam\Track:=track0;
	   ArcL OSPiv2Fwrap_H2, v100, smJK, wdJK1\Weave:=wv0, z1, tWeldGun\WObj:=wobj_PivCam\Track:=track0;
	   ArcL OSPiv2Fwrap_H3, v100, smJK, wdJK1\Weave:=wvJK, z1, tWeldGun\WObj:=wobj_PivCam\Track:=track0;
	   !ArcL OSPiv2Fwrap_H4, v100, smJK, wdJK1\Weave:=wvJK, z1, tWeldGun\WObj:=wobj_PivCam\Track:=track0;
	   ArcLEnd Offs(OSPiv2Fwrap_H4,-10,0,0), v100, smJK, wdJK\Weave:=wvJK, z1, tWeldGun\WObj:=wobj_PivCam\Track:=trLM10hiteonly;
	   PDispOff;
       MoveL RelTool(OSPiv2Fwrap_H4,0,0,-100), V500, z5, tWeldGun\WObj:=wobj_PivCam;
       MoveL RelTool(OSPiv2Fwrap_H4,0,0,-600), V500, z5, tWeldGun\WObj:=wobj_PivCam;
       MoveL Offs(OSPiv2Fwrap_H4,0,-600,-800), V500, z5, tWeldGun\WObj:=wobj_PivCam;
	   MoveJ pjthomeSTA1zero, vCellSpeed, fine, tWeldGun\WObj:=wobj0;
       HIJKLMNOP:
    ENDPROC

!!!!!!!!!!!!!!!!!!!!!!!!!!!!!!!!!!!!!!!!!!!!!!!!!!!!
!!!!!!!!!!!!!!!!!!!!!!!!!!!!!!!!!!!!!!!!!!!!!!!!!!!!
    PROC SET_ANCHOR_SRCH()
    !!!!!!!!!!!THIS PROC HAS BEEN partially modified (6099135,6802707,6862141,6089394, 6850291,689234) these numbers MODIFIED FOR SEARCHING ANCHORS TOTALLY WITH THE NOZZLE 02-05-18!!!!!!!
!!!!!!!!!!!!!!!!REVISED 03-16-18 to add anchor_back X searches!!!!!
IF ANCHOR_USED = 689234 THEN
	! ANCHOR "Y BACK" SEARCH  L & R
	SP_AGBY_E.trans.x := (FAMILY_GX.trans.x + NOZZLE_RADIUS + SIDEPLATE + 107 ); ! 44 Represents the middle between the sideplate and anchor lug
	SP_AGBY_E.trans.y := -13.5;	!(yeager changed it 12-02-17)
	SP_AGBY_E.trans.z := -48.5; !(yeager changed it 12-02-17)

	SP_AGBY_S.trans.x := (FAMILY_GX.trans.x + NOZZLE_RADIUS + SIDEPLATE + 107 );
	SP_AGBY_S.trans.y := -53.5; !(yeager changed it 12-02-17)
	SP_AGBY_S.trans.z := -48.5; !(yeager changed it 12-02-17)

	SP_AHBY_E.trans.x := (FAMILY_HX.trans.x - NOZZLE_RADIUS - SIDEPLATE - 107 ); ! 44 Represents the middle between the sideplate and anchor lug
	SP_AHBY_E.trans.y := -13.5; !(yeager changed it 12-02-17)
	SP_AHBY_E.trans.z := -48.5; !(yeager changed it 12-02-17)

	SP_AHBY_S.trans.x := (FAMILY_HX.trans.x - NOZZLE_RADIUS - SIDEPLATE - 107 );
	SP_AHBY_S.trans.y := -53.5; !(yeager changed it 12-02-17)
	SP_AHBY_S.trans.z := -48.5;	!(yeager changed it 12-02-17)

IF WOTOX < 1300 THEN


  	! ANCHOR "Y FRONT" SEARCH  L & R (short)
	SP_AGFY_E.trans.x := (FAMILY_GX.trans.x + NOZZLE_RADIUS + SIDEPLATE + 56.75 ); !yeager changed it 12-04-17...was 106.75
	SP_AGFY_E.trans.y := 13.5;	!(yeager changed it 12-02-17)
	SP_AGFY_E.trans.z := 9;	!(yeager changed it 12-02-17)

	SP_AGFY_S.trans.x := (FAMILY_GX.trans.x + NOZZLE_RADIUS + SIDEPLATE + 56.75 ); !yeager changed it 12-04-17...was 106.75
	SP_AGFY_S.trans.y := 53.5;	!(yeager changed it 12-02-17)
	SP_AGFY_S.trans.z := 9;	!(yeager changed it 12-02-17)

	SP_AHFY_E.trans.x := (FAMILY_HX.trans.x - NOZZLE_RADIUS - SIDEPLATE - 56.75 ); !yeager changed it 12-04-17...was 106.75
	SP_AHFY_E.trans.y := 13.5;	!(yeager changed it 12-02-17)
	SP_AHFY_E.trans.z := 9;	!(yeager changed it 12-02-17)

	SP_AHFY_S.trans.x := (FAMILY_HX.trans.x - NOZZLE_RADIUS - SIDEPLATE - 56.75 ); !yeager changed it 12-04-17...was 106.75
	SP_AHFY_S.trans.y := 53.5;	!(yeager changed it 12-02-17)
	SP_AHFY_S.trans.z := 9;	!(yeager changed it 12-02-17)

ELSE

  	! ANCHOR "Y FRONT" SEARCH  L & R (long)
	SP_AGFY_E.trans.x := (FAMILY_GX.trans.x + NOZZLE_RADIUS + SIDEPLATE + 106.75 ); !yeager changed it 12-04-17...was 106.75
	SP_AGFY_E.trans.y := 13.5;	!(yeager changed it 12-02-17)
	SP_AGFY_E.trans.z := -48.5;	!(yeager changed it 12-02-17)

	SP_AGFY_S.trans.x := (FAMILY_GX.trans.x + NOZZLE_RADIUS + SIDEPLATE + 106.75 ); !yeager changed it 12-04-17...was 106.75
	SP_AGFY_S.trans.y := 53.5;	!(yeager changed it 12-02-17)
	SP_AGFY_S.trans.z := -48.5;	!(yeager changed it 12-02-17)

	SP_AHFY_E.trans.x := (FAMILY_HX.trans.x - NOZZLE_RADIUS - SIDEPLATE - 106.75 ); !yeager changed it 12-04-17...was 106.75
	SP_AHFY_E.trans.y := 13.5;	!(yeager changed it 12-02-17)
	SP_AHFY_E.trans.z := -48.5;	!(yeager changed it 12-02-17)

	SP_AHFY_S.trans.x := (FAMILY_HX.trans.x - NOZZLE_RADIUS - SIDEPLATE - 106.75 ); !yeager changed it 12-04-17...was 106.75
	SP_AHFY_S.trans.y := 53.5;	!(yeager changed it 12-02-17)
	SP_AHFY_S.trans.z := -48.5;	!(yeager changed it 12-02-17)

ENDIF

    ! ANCHOR BACK  "Z" SEARCH L & R
	SP_AGBZ_E.trans.x := (FAMILY_GX.trans.x + NOZZLE_RADIUS + SIDEPLATE + 102.5 ); ! 102.5 Represents distance from the sideplate to the center of the Anchor lug
	SP_AGBZ_E.trans.y := 75;
	SP_AGBZ_E.trans.z := NOZZLE_RADIUS;

	SP_AGBZ_S.trans.x := (FAMILY_GX.trans.x + NOZZLE_RADIUS + SIDEPLATE + 102.5 );
	SP_AGBZ_S.trans.y := 75;
	SP_AGBZ_S.trans.z := NOZZLE_RADIUS + 30;

	SP_AHBZ_E.trans.x := (FAMILY_HX.trans.x - NOZZLE_RADIUS - SIDEPLATE - 102.5 ); ! 102.5 Represents distance from the sideplate to the center of the Anchor lug
	SP_AHBZ_E.trans.y := 75;
	SP_AHBZ_E.trans.z := NOZZLE_RADIUS;

	SP_AHBZ_S.trans.x := (FAMILY_HX.trans.x - NOZZLE_RADIUS - SIDEPLATE - 102.5 );
	SP_AHBZ_S.trans.y := 75;
	SP_AHBZ_S.trans.z := NOZZLE_RADIUS + 30;

        ! ANCHOR FRONT  "Z" SEARCH L & R
	SP_AGFZ_E.trans.x := (FAMILY_GX.trans.x + NOZZLE_RADIUS + SIDEPLATE + 102.5 ); ! 102.5 Represents distance from the sideplate to the center of the Anchor lug
	SP_AGFZ_E.trans.y := -75;
	SP_AGFZ_E.trans.z := NOZZLE_RADIUS;

	SP_AGFZ_S.trans.x := (FAMILY_GX.trans.x + NOZZLE_RADIUS + SIDEPLATE + 102.5 );
	SP_AGFZ_S.trans.y := -75;
	SP_AGFZ_S.trans.z := NOZZLE_RADIUS + 30;

	SP_AHFZ_E.trans.x := (FAMILY_HX.trans.x - NOZZLE_RADIUS - SIDEPLATE - 102.5 ); ! 102.5 Represents distance from the sideplate to the center of the Anchor lug
	SP_AHFZ_E.trans.y := -75;
	SP_AHFZ_E.trans.z := NOZZLE_RADIUS;

	SP_AHFZ_S.trans.x := (FAMILY_HX.trans.x - NOZZLE_RADIUS - SIDEPLATE - 102.5 );
	SP_AHFZ_S.trans.y := -75;
	SP_AHFZ_S.trans.z := NOZZLE_RADIUS + 30;

    ! ANCHOR BACK "X" SEARCH G & H

	SP_GX_E.trans.x := (FAMILY_GX.trans.x + (NOZZLE_RADIUS*2) + SIDEPLATE  );
	SP_GX_E.trans.y := 0;
	SP_GX_E.trans.z := 35;

	SP_GX_S.trans.x := (FAMILY_GX.trans.x + (NOZZLE_RADIUS*2) + SIDEPLATE + 30 ); !30 Represents generic search length
	SP_GX_S.trans.y := 0;
	SP_GX_S.trans.z := 35;

	SP_HX_E.trans.x := (FAMILY_HX.trans.x - (NOZZLE_RADIUS*2) - SIDEPLATE  );
	SP_HX_E.trans.y := 0;
	SP_HX_E.trans.z := 35;

	SP_HX_S.trans.x := (FAMILY_HX.trans.x - (NOZZLE_RADIUS*2) - SIDEPLATE - 30 ); !30 Represents generic search length
	SP_HX_S.trans.y := 0;
	SP_HX_S.trans.z := 35;


        ! ANCHOR FRONT  "X" SEARCH G & H
	SP_AGFX_E.trans.x := FAMILY_GX.trans.x  + SIDEPLATE + (2 * NOZZLE_RADIUS); ! 40 Represents Search Distance
	SP_AGFX_E.trans.y := -50;
	SP_AGFX_E.trans.z := NOZZLE_RADIUS + 30;

	SP_AGFX_S.trans.x := FAMILY_GX.trans.x  + SIDEPLATE + (2 * NOZZLE_RADIUS) + 40;
	SP_AGFX_S.trans.y := -50;
	SP_AGFX_S.trans.z := NOZZLE_RADIUS + 30;

!!!!!!!!!!!!!!!!!!!!!!!!!!!!!!!!!!!!!!!!!!!!
	SP_AHFX_E.trans.x := FAMILY_HX.trans.x - SIDEPLATE - (2 * NOZZLE_RADIUS); ! 40 Represents Search Distance
	SP_AHFX_E.trans.y := -50;
	SP_AHFX_E.trans.z := NOZZLE_RADIUS + 30;

	SP_AHFX_S.trans.x := FAMILY_HX.trans.x - SIDEPLATE - (2 * NOZZLE_RADIUS) - 40;
	SP_AHFX_S.trans.y := -50;
	SP_AHFX_S.trans.z := NOZZLE_RADIUS + 30;


ELSE IF ANCHOR_USED = 6099135 THEN

!!!!!!!MODIFIED THESE VALUES for 18H ANCHORS 02-05-18!!!!!!!!!!!
	! ANCHOR "Y TOP" SEARCH  L & R
	SP_AGBY_E.trans.x := (FAMILY_GX.trans.x + NOZZLE_RADIUS + SIDEPLATE + 59 ); ! 36.5 Represents the middle between the sideplate and anchor lug
	SP_AGBY_E.trans.y := -13.5;		!50.8 REPRESENTS THICKNESS OF THE ANCHOR
	SP_AGBY_E.trans.z := -50 ;		! Represents distance from lug tangent to anchor body

	SP_AGBY_S.trans.x := (FAMILY_GX.trans.x + NOZZLE_RADIUS + SIDEPLATE + 59 );
	SP_AGBY_S.trans.y := -53.5;		!50.8 REPRESENTS THICKNESS OF THE ANCHOR
	SP_AGBY_S.trans.z := -50 ;		! Represents distance from lug tangent to anchor body


	SP_AHBY_E.trans.x := (FAMILY_HX.trans.x - NOZZLE_RADIUS - SIDEPLATE - 59 ); ! 36.5 Represents the middle between the sideplate and anchor lug
	SP_AHBY_E.trans.y := -13.5;	!50.8 REPRESENTS THICKNESS OF THE ANCHOR
	SP_AHBY_E.trans.z := -50 ;	! Represents distance from lug tangent to anchor body

	SP_AHBY_S.trans.x := (FAMILY_HX.trans.x - NOZZLE_RADIUS - SIDEPLATE - 59 );
	SP_AHBY_S.trans.y := -53.5;	!50.8 REPRESENTS THICKNESS OF THE ANCHOR
	SP_AHBY_S.trans.z := -50 ;	! Represents distance from lug tangent to anchor body
!!!!!!!end of MODIFIED THESE VALUES for 18H ANCHORS 02-05-18!!!!!!!!!!!

	! ANCHOR "Z" SEARCH L & R
	SP_AGBZ_E.trans.x := (FAMILY_GX.trans.x + NOZZLE_RADIUS + SIDEPLATE + 58.25 ); ! 58.25 Represents distance from the sideplate to the center of the Anchor lug
	SP_AGBZ_E.trans.y := 60;    ! Represents roughly the wire STICK_OUT (TCP) to be below the flat bottom of the anchor
	SP_AGBZ_E.trans.z := NOZZLE_RADIUS;

	SP_AGBZ_S.trans.x := (FAMILY_GX.trans.x + NOZZLE_RADIUS + SIDEPLATE + 58.25 );
	SP_AGBZ_S.trans.y := 60;     ! Represents roughly the wire STICK_OUT (TCP) to be below the flat bottom of the anchor
	SP_AGBZ_S.trans.z := NOZZLE_RADIUS + 30;	!!  just a search length

	SP_AHBZ_E.trans.x := (FAMILY_HX.trans.x - NOZZLE_RADIUS - SIDEPLATE - 58.25 ); ! 58.25 Represents distance from the sideplate to the center of the Anchor lug
	SP_AHBZ_E.trans.y := 60;	! Represents roughly the wire STICK_OUT (TCP) to be below the flat bottom of the anchor
	SP_AHBZ_E.trans.z := NOZZLE_RADIUS;

	SP_AHBZ_S.trans.x := (FAMILY_HX.trans.x - NOZZLE_RADIUS - SIDEPLATE - 58.25 );
	SP_AHBZ_S.trans.y := 60;	! Represents roughly the wire STICK_OUT (TCP) to be below the flat bottom of the anchor
	SP_AHBZ_S.trans.z := NOZZLE_RADIUS + 30; !!  just a search length

IF WOTOX < 1200 THEN


    ! ANCHOR "Y BOTTOM" SEARCH  L & R
!!!!!!!MODIFIED THESE VALUES for 18H ANCHORS 02-05-18!!!!!!!!!!!
    SP_AGFY_E.trans.x := -65;
    SP_AGFY_E.trans.y := 13.5;		! NOZZLE_RADIUS REPRESENTS the nozzle flush on the casting
	SP_AGFY_E.trans.z := -170 ;		! Represents distance from lug tangent to anchor body

	SP_AGFY_S.trans.x := -65;
	SP_AGFY_S.trans.y := 53.5;		! NOZZLE_RADIUS REPRESENTS the nozzle flush on the casting
	SP_AGFY_S.trans.z := -170 ;		! Represents distance from lug tangent to anchor body

    SP_AHFY_E.trans.x := 65;
	SP_AHFY_E.trans.y := 13.5;	! NOZZLE_RADIUS REPRESENTS the nozzle flush on the casing
	SP_AHFY_E.trans.z := -170 ;	! Represents distance from lug tangent to anchor body

	SP_AHFY_S.trans.x := 65;
	SP_AHFY_S.trans.y := 53.5;		! NOZZLE_RADIUS REPRESENTS the nozzle flush on the casting
	SP_AHFY_S.trans.z := -170 ;		! Represents distance from lug tangent to anchor body

    ! ANCHOR "Z BOTTOM" SEARCH L & R
!!!!!!!end of MODIFIED THESE VALUES for 18H ANCHORS 02-05-18!!!!!!!!!!!

    SP_AGFZ_E.trans.x := (FAMILY_GX.trans.x + NOZZLE_RADIUS + SIDEPLATE + 58.25 ); ! 72.5 Represents the distance from the sideplate to the center of the anchor lug
	SP_AGFZ_E.trans.y := -65;    ! Represents roughly the wire STICK_OUT (TCP) to be below the flat bottom of the anchor
	SP_AGFZ_E.trans.z := NOZZLE_RADIUS;

	SP_AGFZ_S.trans.x := (FAMILY_GX.trans.x + NOZZLE_RADIUS + SIDEPLATE + 58.25 ); ! 72.5 Represents the distance from the sideplate to the center of the anchor lug
	SP_AGFZ_S.trans.y := -65;     ! Represents roughly the wire STICK_OUT (TCP) to be below the flat bottom of the anchor
	SP_AGFZ_S.trans.z := NOZZLE_RADIUS + 30;	!!  just a search length

	SP_AHFZ_E.trans.x := (FAMILY_HX.trans.x - NOZZLE_RADIUS - SIDEPLATE - 58.25 ); ! 72.5 Represents the distance from the sideplate to the center of the anchor lug
	SP_AHFZ_E.trans.y := -65;	! Represents roughly the wire STICK_OUT (TCP) to be below the flat bottom of the anchor
	SP_AHFZ_E.trans.z := NOZZLE_RADIUS;

	SP_AHFZ_S.trans.x := (FAMILY_HX.trans.x - NOZZLE_RADIUS - SIDEPLATE - 58.25 ); ! 72.5 Represents the distance from the sideplate to the center of the anchor lug
	SP_AHFZ_S.trans.y := -65;	! Represents roughly the wire STICK_OUT (TCP) to be below the flat bottom of the anchor
	SP_AHFZ_S.trans.z := NOZZLE_RADIUS + 30; !!  just a search length


 ELSE


    ! ANCHOR "Y BOTTOM" SEARCH  L & R
!!!!!!!MODIFIED THESE VALUES for 18H ANCHORS 02-05-18!!!!!!!!!!!
    SP_AGFY_E.trans.x := (FAMILY_GX.trans.x + NOZZLE_RADIUS + SIDEPLATE + 59 ); ! 36.5 Represents the distance from the sideplate to the center of the anchor lug
	SP_AGFY_E.trans.y := 13.5;		! NOZZLE_RADIUS REPRESENTS the nozzle flush on the casting
	SP_AGFY_E.trans.z := -50 ;		! Represents distance from lug tangent to anchor body

	SP_AGFY_S.trans.x := (FAMILY_GX.trans.x + NOZZLE_RADIUS + SIDEPLATE + 59 );  ! 36.5 Represents the distance from the sideplate to the center of the anchor lug
	SP_AGFY_S.trans.y := 53.5;		! NOZZLE_RADIUS REPRESENTS the nozzle flush on the casting
	SP_AGFY_S.trans.z := -50 ;		! Represents distance from lug tangent to anchor body

    SP_AHFY_E.trans.x := (FAMILY_HX.trans.x - NOZZLE_RADIUS - SIDEPLATE - 59 ); !36.5 Represents the distance from the sideplate to the center of the anchor lug
	SP_AHFY_E.trans.y := 13.5;	! NOZZLE_RADIUS REPRESENTS the nozzle flush on the casing
	SP_AHFY_E.trans.z := -50 ;	! Represents distance from lug tangent to anchor body

	SP_AHFY_S.trans.x := (FAMILY_HX.trans.x - NOZZLE_RADIUS - SIDEPLATE - 59 );  ! 36.5 Represents the distance from the sideplate to the center of the anchor lug
	SP_AHFY_S.trans.y := 53.5;		! NOZZLE_RADIUS REPRESENTS the nozzle flush on the casting
	SP_AHFY_S.trans.z := -50 ;		! Represents distance from lug tangent to anchor body
	! ANCHOR "Z BOTTOM" SEARCH L & R
!!!!!!!end of MODIFIED THESE VALUES for 18H ANCHORS 02-05-18!!!!!!!!!!!

    SP_AGFZ_E.trans.x := (FAMILY_GX.trans.x + NOZZLE_RADIUS + SIDEPLATE + 58.25 ); ! 72.5 Represents the distance from the sideplate to the center of the anchor lug
	SP_AGFZ_E.trans.y := -65;    ! Represents roughly the wire STICK_OUT (TCP) to be below the flat bottom of the anchor
	SP_AGFZ_E.trans.z := NOZZLE_RADIUS;

	SP_AGFZ_S.trans.x := (FAMILY_GX.trans.x + NOZZLE_RADIUS + SIDEPLATE + 58.25 ); ! 72.5 Represents the distance from the sideplate to the center of the anchor lug
	SP_AGFZ_S.trans.y := -65;     ! Represents roughly the wire STICK_OUT (TCP) to be below the flat bottom of the anchor
	SP_AGFZ_S.trans.z := NOZZLE_RADIUS + 30;	!!  just a search length

	SP_AHFZ_E.trans.x := (FAMILY_HX.trans.x - NOZZLE_RADIUS - SIDEPLATE - 58.25 ); ! 72.5 Represents the distance from the sideplate to the center of the anchor lug
	SP_AHFZ_E.trans.y := -65;	! Represents roughly the wire STICK_OUT (TCP) to be below the flat bottom of the anchor
	SP_AHFZ_E.trans.z := NOZZLE_RADIUS;

	SP_AHFZ_S.trans.x := (FAMILY_HX.trans.x - NOZZLE_RADIUS - SIDEPLATE - 58.25 ); ! 72.5 Represents the distance from the sideplate to the center of the anchor lug
	SP_AHFZ_S.trans.y := -65;	! Represents roughly the wire STICK_OUT (TCP) to be below the flat bottom of the anchor
	SP_AHFZ_S.trans.z := NOZZLE_RADIUS + 30; !!  just a search length

ENDIF

	! ANCHOR BACK "X" SEARCH G & H

	SP_GX_E.trans.x := (FAMILY_GX.trans.x + (NOZZLE_RADIUS*2) + SIDEPLATE  );
	SP_GX_E.trans.y := 0;
	SP_GX_E.trans.z := 25;  ! distance behind the lug of the anchor

	SP_GX_S.trans.x := (FAMILY_GX.trans.x + (NOZZLE_RADIUS*2) + SIDEPLATE + 30 ); !30 Represents generic search length
	SP_GX_S.trans.y := 0;
	SP_GX_S.trans.z := 25;	! distance behind the lug of the anchor

	SP_HX_E.trans.x := (FAMILY_HX.trans.x - (NOZZLE_RADIUS*2) - SIDEPLATE  );
	SP_HX_E.trans.y := 0;
	SP_HX_E.trans.z := 25;	! distance behind the lug of the anchor

	SP_HX_S.trans.x := (FAMILY_HX.trans.x - (NOZZLE_RADIUS*2) - SIDEPLATE - 30 ); !30 Represents generic search length
	SP_HX_S.trans.y := 0;
	SP_HX_S.trans.z := 25;		! distance behind the lug of the anchor


        ! ANCHOR FRONT  "X" SEARCH G & H
	SP_AGFX_E.trans.x := FAMILY_GX.trans.x  + SIDEPLATE + (2 * NOZZLE_RADIUS); ! 40 Represents Search Distance
	SP_AGFX_E.trans.y := -50;
	SP_AGFX_E.trans.z := NOZZLE_RADIUS + 30;

	SP_AGFX_S.trans.x := FAMILY_GX.trans.x  + SIDEPLATE + (2 * NOZZLE_RADIUS) + 40;
	SP_AGFX_S.trans.y := -50;
	SP_AGFX_S.trans.z := NOZZLE_RADIUS + 30;

!!!!!!!!!!!!!!!!!!!!!!!!!!!!!!!!!!!!!!!!!!!!
	SP_AHFX_E.trans.x := FAMILY_HX.trans.x - SIDEPLATE - (2 * NOZZLE_RADIUS); ! 40 Represents Search Distance
	SP_AHFX_E.trans.y := -50;
	SP_AHFX_E.trans.z := NOZZLE_RADIUS + 30;

	SP_AHFX_S.trans.x := FAMILY_HX.trans.x - SIDEPLATE - (2 * NOZZLE_RADIUS) - 40;
	SP_AHFX_S.trans.y := -50;
	SP_AHFX_S.trans.z := NOZZLE_RADIUS + 30;


ELSE IF ANCHOR_USED = 6089394 THEN

    !!!!!!!!!!!!!!!THIS 6039394 group HAS values changed FOR A NOZZLE SEARCH TEST 11-29-17!!!!!!!!

    IF WOTOX < 1400 THEN
     ! for short wotox!
	SP_AGBY_E.trans.x := (FAMILY_GX.trans.x + NOZZLE_RADIUS + SIDEPLATE + 72.5 ); ! 72.5 Represents the distance from the sideplate to the center of the anchor lug
	SP_AGBY_E.trans.y := -13.5;		! NOZZLE_RADIUS REPRESENTS the nozzle flush on the casing (yeager changed it 11-27-17)
	SP_AGBY_E.trans.z := -130 ;		! Represents distance from lug tangent to anchor body (yeager changed it 11-27-17)

	SP_AGBY_S.trans.x := (FAMILY_GX.trans.x + NOZZLE_RADIUS + SIDEPLATE + 72.5 );  ! 72.5 Represents the distance from the sideplate to the center of the anchor lug
	SP_AGBY_S.trans.y := -53.5;		! NOZZLE_RADIUS REPRESENTS the nozzle flush on the casing (yeager changed it 11-27-17)
	SP_AGBY_S.trans.z := -130 ;		! Represents distance from lug tangent to anchor body (yeager changed it 11-27-17)

    SP_AHBY_E.trans.x := (FAMILY_HX.trans.x - NOZZLE_RADIUS - SIDEPLATE - 72.5 ); !72.5 Represents the distance from the sideplate to the center of the anchor lug
	SP_AHBY_E.trans.y := -13.5;	! NOZZLE_RADIUS REPRESENTS the nozzle flush on the casing  (yeager changed it 11-27-17)
	SP_AHBY_E.trans.z := -130 ;	! Represents distance from lug tangent to anchor body	(yeager changed it 11-27-17)

	SP_AHBY_S.trans.x := (FAMILY_HX.trans.x - NOZZLE_RADIUS - SIDEPLATE - 72.5 );  ! 72.5 Represents the distance from the sideplate to the center of the anchor lug
	SP_AHBY_S.trans.y := -53.5;		! NOZZLE_RADIUS REPRESENTS the nozzle flush on the casing (yeager changed it 11-27-17)
	SP_AHBY_S.trans.z := -130 ;		! Represents distance from lug tangent to anchor body	(yeager changed it 11-27-17)

    ELSE

    ! for long wotox
	SP_AGBY_E.trans.x := (FAMILY_GX.trans.x + NOZZLE_RADIUS + SIDEPLATE + 72.5 ); ! 72.5 Represents the distance from the sideplate to the center of the anchor lug
	SP_AGBY_E.trans.y := -13.5;		! NOZZLE_RADIUS REPRESENTS the nozzle flush on the casing (yeager changed it 11-27-17)
	SP_AGBY_E.trans.z := -5 ;		! Represents distance from lug tangent to anchor body (yeager changed it 11-27-17)

	SP_AGBY_S.trans.x := (FAMILY_GX.trans.x + NOZZLE_RADIUS + SIDEPLATE + 72.5 );  ! 72.5 Represents the distance from the sideplate to the center of the anchor lug
	SP_AGBY_S.trans.y := -53.5;		! NOZZLE_RADIUS REPRESENTS the nozzle flush on the casing (yeager changed it 11-27-17)
	SP_AGBY_S.trans.z := -5 ;		! Represents distance from lug tangent to anchor body (yeager changed it 11-27-17)

    SP_AHBY_E.trans.x := (FAMILY_HX.trans.x - NOZZLE_RADIUS - SIDEPLATE - 72.5 ); !72.5 Represents the distance from the sideplate to the center of the anchor lug
	SP_AHBY_E.trans.y := -13.5;	! NOZZLE_RADIUS REPRESENTS the nozzle flush on the casing  (yeager changed it 11-27-17)
	SP_AHBY_E.trans.z := -5 ;	! Represents distance from lug tangent to anchor body	(yeager changed it 11-27-17)

	SP_AHBY_S.trans.x := (FAMILY_HX.trans.x - NOZZLE_RADIUS - SIDEPLATE - 72.5 );  ! 72.5 Represents the distance from the sideplate to the center of the anchor lug
	SP_AHBY_S.trans.y := -53.5;		! NOZZLE_RADIUS REPRESENTS the nozzle flush on the casing (yeager changed it 11-27-17)
	SP_AHBY_S.trans.z := -5 ;		! Represents distance from lug tangent to anchor body	(yeager changed it 11-27-17)


  ENDIF

    ! ANCHOR "Z TOP" SEARCH L & R
	SP_AGBZ_E.trans.x := (FAMILY_GX.trans.x + NOZZLE_RADIUS + SIDEPLATE + 72.5 ); ! 72.5 Represents the distance from the sideplate to the center of the anchor lug
	SP_AGBZ_E.trans.y := 75;    ! Represents roughly the wire STICK_OUT (TCP) to be below the flat bottom of the anchor
	SP_AGBZ_E.trans.z := NOZZLE_RADIUS;

	SP_AGBZ_S.trans.x := (FAMILY_GX.trans.x + NOZZLE_RADIUS + SIDEPLATE + 72.5 ); ! 72.5 Represents the distance from the sideplate to the center of the anchor lug
	SP_AGBZ_S.trans.y := 75;     ! Represents roughly the wire STICK_OUT (TCP) to be below the flat bottom of the anchor
	SP_AGBZ_S.trans.z := NOZZLE_RADIUS + 30;	!!  just a search length

	SP_AHBZ_E.trans.x := (FAMILY_HX.trans.x - NOZZLE_RADIUS - SIDEPLATE - 72.5 ); ! 72.5 Represents the distance from the sideplate to the center of the anchor lug
	SP_AHBZ_E.trans.y := 75;	! Represents roughly the wire STICK_OUT (TCP) to be below the flat bottom of the anchor
	SP_AHBZ_E.trans.z := NOZZLE_RADIUS;

	SP_AHBZ_S.trans.x := (FAMILY_HX.trans.x - NOZZLE_RADIUS - SIDEPLATE - 72.5 ); ! 72.5 Represents the distance from the sideplate to the center of the anchor lug
	SP_AHBZ_S.trans.y := 75;	! Represents roughly the wire STICK_OUT (TCP) to be below the flat bottom of the anchor
	SP_AHBZ_S.trans.z := NOZZLE_RADIUS + 30; !!  just a search length


 IF WOTOX < 1400 THEN

  	! points at tip (for short wotox parts)
	SP_AGFY_E.trans.x := (FAMILY_GX.trans.x + NOZZLE_RADIUS + SIDEPLATE + 72.5 ); ! 72.5 Represents the distance from the sideplate to the center of the anchor lug
	SP_AGFY_E.trans.y := 13.5;		! NOZZLE_RADIUS REPRESENTS the nozzle flush on the casting (yeager changed it 11-27-17)
	SP_AGFY_E.trans.z := -130 ;		! Represents distance from lug tangent to anchor body (yeager changed it 11-27-17)

	SP_AGFY_S.trans.x := (FAMILY_GX.trans.x + NOZZLE_RADIUS + SIDEPLATE + 72.5 );  ! 72.5 Represents the distance from the sideplate to the center of the anchor lug
	SP_AGFY_S.trans.y := 53.5;		! NOZZLE_RADIUS REPRESENTS the nozzle flush on the casting (yeager changed it 11-27-17)
	SP_AGFY_S.trans.z := -130 ;		! Represents distance from lug tangent to anchor body (yeager changed it 11-27-17)

    SP_AHFY_E.trans.x := (FAMILY_HX.trans.x - NOZZLE_RADIUS - SIDEPLATE - 72.5 ); !72.5 Represents the distance from the sideplate to the center of the anchor lug
	SP_AHFY_E.trans.y := 13.5;	! NOZZLE_RADIUS REPRESENTS the nozzle flush on the casing (yeager changed it 11-27-17)
	SP_AHFY_E.trans.z := -130 ;	! Represents distance from lug tangent to anchor body	(yeager changed it 11-27-17)

	SP_AHFY_S.trans.x := (FAMILY_HX.trans.x - NOZZLE_RADIUS - SIDEPLATE - 72.5 );  ! 72.5 Represents the distance from the sideplate to the center of the anchor lug
	SP_AHFY_S.trans.y := 53.5;		! NOZZLE_RADIUS REPRESENTS the nozzle flush on the casting (yeager changed it 11-27-17)
	SP_AHFY_S.trans.z := -130 ;		! Represents distance from lug tangent to anchor body (yeager changed it 11-27-17)

ELSE
	! ANCHOR "Y BOTTOM" SEARCH  L & R
	SP_AGFY_E.trans.x := (FAMILY_GX.trans.x + NOZZLE_RADIUS + SIDEPLATE + 72.5 ); ! 72.5 Represents the distance from the sideplate to the center of the anchor lug
	SP_AGFY_E.trans.y := 13.5;		! NOZZLE_RADIUS REPRESENTS the nozzle flush on the casting (yeager changed it 11-27-17)
	SP_AGFY_E.trans.z := -5 ;		! Represents distance from lug tangent to anchor body (yeager changed it 11-27-17)

	SP_AGFY_S.trans.x := (FAMILY_GX.trans.x + NOZZLE_RADIUS + SIDEPLATE + 72.5 );  ! 72.5 Represents the distance from the sideplate to the center of the anchor lug
	SP_AGFY_S.trans.y := 53.5;		! NOZZLE_RADIUS REPRESENTS the nozzle flush on the casting (yeager changed it 11-27-17)
	SP_AGFY_S.trans.z := -5 ;		! Represents distance from lug tangent to anchor body (yeager changed it 11-27-17)

    SP_AHFY_E.trans.x := (FAMILY_HX.trans.x - NOZZLE_RADIUS - SIDEPLATE - 72.5 ); !72.5 Represents the distance from the sideplate to the center of the anchor lug
	SP_AHFY_E.trans.y := 13.5;	! NOZZLE_RADIUS REPRESENTS the nozzle flush on the casing (yeager changed it 11-27-17)
	SP_AHFY_E.trans.z := -5 ;	! Represents distance from lug tangent to anchor body	(yeager changed it 11-27-17)

	SP_AHFY_S.trans.x := (FAMILY_HX.trans.x - NOZZLE_RADIUS - SIDEPLATE - 72.5 );  ! 72.5 Represents the distance from the sideplate to the center of the anchor lug
	SP_AHFY_S.trans.y := 53.5;		! NOZZLE_RADIUS REPRESENTS the nozzle flush on the casting (yeager changed it 11-27-17)
	SP_AHFY_S.trans.z := -5 ;		! Represents distance from lug tangent to anchor body (yeager changed it 11-27-17)

 ENDIF
    ! ANCHOR "Z BOTTOM" SEARCH L & R
    SP_AGFZ_E.trans.x := (FAMILY_GX.trans.x + NOZZLE_RADIUS + SIDEPLATE + 72.5 ); ! 72.5 Represents the distance from the sideplate to the center of the anchor lug
	SP_AGFZ_E.trans.y := -90;    ! Represents roughly the wire STICK_OUT (TCP) to be below the flat bottom of the anchor
	SP_AGFZ_E.trans.z := NOZZLE_RADIUS;

	SP_AGFZ_S.trans.x := (FAMILY_GX.trans.x + NOZZLE_RADIUS + SIDEPLATE + 72.5 ); ! 72.5 Represents the distance from the sideplate to the center of the anchor lug
	SP_AGFZ_S.trans.y := -90;     ! Represents roughly the wire STICK_OUT (TCP) to be below the flat bottom of the anchor
	SP_AGFZ_S.trans.z := NOZZLE_RADIUS + 30;	!!  just a search length

	SP_AHFZ_E.trans.x := (FAMILY_HX.trans.x - NOZZLE_RADIUS - SIDEPLATE - 72.5 ); ! 72.5 Represents the distance from the sideplate to the center of the anchor lug
	SP_AHFZ_E.trans.y := -90;	! Represents roughly the wire STICK_OUT (TCP) to be below the flat bottom of the anchor
	SP_AHFZ_E.trans.z := NOZZLE_RADIUS;

	SP_AHFZ_S.trans.x := (FAMILY_HX.trans.x - NOZZLE_RADIUS - SIDEPLATE - 72.5 ); ! 72.5 Represents the distance from the sideplate to the center of the anchor lug
	SP_AHFZ_S.trans.y := -90;	! Represents roughly the wire STICK_OUT (TCP) to be below the flat bottom of the anchor
	SP_AHFZ_S.trans.z := NOZZLE_RADIUS + 30; !!  just a search length

	! ANCHOR BACK "X" SEARCH G & H

	SP_GX_E.trans.x := (FAMILY_GX.trans.x + (NOZZLE_RADIUS*2) + SIDEPLATE  );
	SP_GX_E.trans.y := 0;
	SP_GX_E.trans.z := 30;  ! distance behind the lug of the anchor

	SP_GX_S.trans.x := (FAMILY_GX.trans.x + (NOZZLE_RADIUS*2) + SIDEPLATE + 25 ); ! 30 Represents generic search length
	SP_GX_S.trans.y := 0;
	SP_GX_S.trans.z := 30;	! distance behind the lug of the anchor

	SP_HX_E.trans.x := (FAMILY_HX.trans.x - (NOZZLE_RADIUS*2) - SIDEPLATE  );
	SP_HX_E.trans.y := 0;
	SP_HX_E.trans.z := 30;	! distance behind the lug of the anchor

	SP_HX_S.trans.x := (FAMILY_HX.trans.x - (NOZZLE_RADIUS*2) - SIDEPLATE - 25 ); ! 30 Represents generic search length
	SP_HX_S.trans.y := 0;
	SP_HX_S.trans.z := 30;		! distance behind the lug of the anchor


        ! ANCHOR FRONT  "X" SEARCH G & H
	SP_AGFX_E.trans.x := FAMILY_GX.trans.x  + SIDEPLATE + (2 * NOZZLE_RADIUS); ! 40 Represents Search Distance
	SP_AGFX_E.trans.y := -50;
	SP_AGFX_E.trans.z := NOZZLE_RADIUS + 30;

	SP_AGFX_S.trans.x := FAMILY_GX.trans.x  + SIDEPLATE + (2 * NOZZLE_RADIUS) + 40;
	SP_AGFX_S.trans.y := -50;
	SP_AGFX_S.trans.z := NOZZLE_RADIUS + 30;

!!!!!!!!!!!!!!!!!!!!!!!!!!!!!!!!!!!!!!!!!!!!
	SP_AHFX_E.trans.x := FAMILY_HX.trans.x - SIDEPLATE - (2 * NOZZLE_RADIUS); ! 40 Represents Search Distance
	SP_AHFX_E.trans.y := -50;
	SP_AHFX_E.trans.z := NOZZLE_RADIUS + 30;

	SP_AHFX_S.trans.x := FAMILY_HX.trans.x - SIDEPLATE - (2 * NOZZLE_RADIUS) - 40;
	SP_AHFX_S.trans.y := -50;
	SP_AHFX_S.trans.z := NOZZLE_RADIUS + 30;


    ELSE IF ANCHOR_USED = 6850291 THEN
    !!!!!!!!!!!!!!!THIS 6850291 group HAS values changed FOR A NOZZLE SEARCH TEST 12-01-17!!!!!!!!
    !!!!!!!!!!!!!!!added variables for short wotox(<1300) 01-10-18!!!!!!!!
    ! BACK ANCHOR "Y TOP" SEARCH  L & R      wobjHanchor_BACK
	SP_AGBY_E.trans.x := (FAMILY_GX.trans.x + NOZZLE_RADIUS + SIDEPLATE + 101.2 ); ! 101.2 Represents the middle between the sideplate and anchor lug
	SP_AGBY_E.trans.y := -15.5;!(yeager changed it 12-01-17)
	SP_AGBY_E.trans.z := -25 ;!(yeager changed it 12-01-17)

	SP_AGBY_S.trans.x := (FAMILY_GX.trans.x + NOZZLE_RADIUS + SIDEPLATE + 101.2 );
	SP_AGBY_S.trans.y := -50.5;!(yeager changed it 12-01-17)
	SP_AGBY_S.trans.z := -25;!(yeager changed it 12-01-17)

	SP_AHBY_E.trans.x := (FAMILY_HX.trans.x - NOZZLE_RADIUS - SIDEPLATE - 101.2 ); ! 101.2 Represents the middle between the sideplate and anchor lug
	SP_AHBY_E.trans.y := -15.5;!(yeager changed it 12-01-17)
	SP_AHBY_E.trans.z := -25 ;!(yeager changed it 12-01-17)

	SP_AHBY_S.trans.x := (FAMILY_HX.trans.x - NOZZLE_RADIUS - SIDEPLATE - 101.2 );
	SP_AHBY_S.trans.y := -50.5;!(yeager changed it 12-01-17)
	SP_AHBY_S.trans.z := -25 ;!(yeager changed it 12-01-17)


	! BACK ANCHOR "Z" SEARCH L & R	         wobjHanchor_BACK
	SP_AGBZ_E.trans.x := (FAMILY_GX.trans.x + NOZZLE_RADIUS + SIDEPLATE + 101.2 ); ! 101.2 Represents distance from the sideplate to the center of the Anchor lug
	SP_AGBZ_E.trans.y := 102.5;
	SP_AGBZ_E.trans.z := NOZZLE_RADIUS;

	SP_AGBZ_S.trans.x := (FAMILY_GX.trans.x + NOZZLE_RADIUS + SIDEPLATE + 101.2 );
	SP_AGBZ_S.trans.y := 102.5;
	SP_AGBZ_S.trans.z := NOZZLE_RADIUS + 35;

	SP_AHBZ_E.trans.x := (FAMILY_HX.trans.x - NOZZLE_RADIUS - SIDEPLATE - 101.2); ! 101.2 Represents distance from the sideplate to the center of the Anchor lug
	SP_AHBZ_E.trans.y := 102.5;
	SP_AHBZ_E.trans.z := NOZZLE_RADIUS;

	SP_AHBZ_S.trans.x := (FAMILY_HX.trans.x - NOZZLE_RADIUS - SIDEPLATE - 101.2 );
	SP_AHBZ_S.trans.y := 102.5;
	SP_AHBZ_S.trans.z := NOZZLE_RADIUS + 35;

	!ANCHOR BACK "X" SEARCH G & H

	SP_GX_E.trans.x := (FAMILY_GX.trans.x + (NOZZLE_RADIUS*2) + SIDEPLATE  );
	SP_GX_E.trans.y := 0;
	SP_GX_E.trans.z := 30;

	SP_GX_S.trans.x := (FAMILY_GX.trans.x + (NOZZLE_RADIUS*2) + SIDEPLATE + 30 ); !30 Represents generic search length
	SP_GX_S.trans.y := 0;
	SP_GX_S.trans.z := 30;

	SP_HX_E.trans.x := (FAMILY_HX.trans.x - (NOZZLE_RADIUS*2) - SIDEPLATE  );
	SP_HX_E.trans.y := 0;
	SP_HX_E.trans.z := 30;

	SP_HX_S.trans.x := (FAMILY_HX.trans.x - (NOZZLE_RADIUS*2) - SIDEPLATE - 30 ); !30 Represents generic search length
	SP_HX_S.trans.y := 0;
	SP_HX_S.trans.z := 30;


        ! ANCHOR FRONT  "X" SEARCH G & H
	SP_AGFX_E.trans.x := FAMILY_GX.trans.x  + SIDEPLATE + (2 * NOZZLE_RADIUS); ! 40 Represents Search Distance
	SP_AGFX_E.trans.y := -50;
	SP_AGFX_E.trans.z := NOZZLE_RADIUS + 30;

	SP_AGFX_S.trans.x := FAMILY_GX.trans.x  + SIDEPLATE + (2 * NOZZLE_RADIUS) + 40;
	SP_AGFX_S.trans.y := -50;
	SP_AGFX_S.trans.z := NOZZLE_RADIUS + 30;

!!!!!!!!!!!!!!!!!!!!!!!!!!!!!!!!!!!!!!!!!!!!
	SP_AHFX_E.trans.x := FAMILY_HX.trans.x - SIDEPLATE - (2 * NOZZLE_RADIUS); ! 40 Represents Search Distance
	SP_AHFX_E.trans.y := -50;
	SP_AHFX_E.trans.z := NOZZLE_RADIUS + 30;

	SP_AHFX_S.trans.x := FAMILY_HX.trans.x - SIDEPLATE - (2 * NOZZLE_RADIUS) - 40;
	SP_AHFX_S.trans.y := -50;
	SP_AHFX_S.trans.z := NOZZLE_RADIUS + 30;


    !!!!! FRONT  ANCHOR "Z" SEARCH L & R	wobjHanchor_FRONT
	SP_AGFZ_E.trans.x := (FAMILY_GX.trans.x + NOZZLE_RADIUS + SIDEPLATE + 101.2 ); ! 101.2 Represents distance from the sideplate to the center of the Anchor lug
	SP_AGFZ_E.trans.y := -102.5;
	SP_AGFZ_E.trans.z := NOZZLE_RADIUS;

	SP_AGFZ_S.trans.x := (FAMILY_GX.trans.x + NOZZLE_RADIUS + SIDEPLATE + 101.2 );
	SP_AGFZ_S.trans.y := -102.5;
	SP_AGFZ_S.trans.z := NOZZLE_RADIUS + 35;

	SP_AHFZ_E.trans.x := (FAMILY_HX.trans.x - NOZZLE_RADIUS - SIDEPLATE - 101.2); ! 101.2 Represents distance from the sideplate to the center of the Anchor lug
	SP_AHFZ_E.trans.y := -102.5;
	SP_AHFZ_E.trans.z := NOZZLE_RADIUS;

	SP_AHFZ_S.trans.x := (FAMILY_HX.trans.x - NOZZLE_RADIUS - SIDEPLATE - 101.2 );
	SP_AHFZ_S.trans.y := -102.5;
	SP_AHFZ_S.trans.z := NOZZLE_RADIUS + 35;

   IF WOTOX < 1300 THEN

  		! FRONT ANCHOR "Y TOP" SEARCH  L & R      wobjHanchor_FRONT
	SP_AGFY_E.trans.x := (FAMILY_GX.trans.x + NOZZLE_RADIUS + SIDEPLATE + 101.2 ); ! 101.2 Represents the middle between the sideplate and anchor lug
	SP_AGFY_E.trans.y := 13.5;!(yeager changed this 01-10-17)
	SP_AGFY_E.trans.z := -150 ;!(yeager changed this 01-10-17)

	SP_AGFY_S.trans.x := (FAMILY_GX.trans.x + NOZZLE_RADIUS + SIDEPLATE + 101.2 );
	SP_AGFY_S.trans.y := 48.5 ;!(yeager changed this 01-10-17)
	SP_AGFY_S.trans.z := -150;!(yeager changed this 01-10-17)

	SP_AHFY_E.trans.x := (FAMILY_HX.trans.x - NOZZLE_RADIUS - SIDEPLATE - 101.2 ); ! 101.2 Represents the middle between the sideplate and anchor lug
	SP_AHFY_E.trans.y := 13.5;!(yeager changed this 01-10-17)
	SP_AHFY_E.trans.z := -150 ;!(yeager changed this 01-10-17)

	SP_AHFY_S.trans.x := (FAMILY_HX.trans.x - NOZZLE_RADIUS - SIDEPLATE - 101.2 );
	SP_AHFY_S.trans.y := 48.5  ;!(yeager changed this 01-10-17)
	SP_AHFY_S.trans.z := -150 ;!(yeager changed this 01-10-17)

ELSE

		! FRONT ANCHOR "Y TOP" SEARCH  L & R      wobjHanchor_FRONT
	SP_AGFY_E.trans.x := (FAMILY_GX.trans.x + NOZZLE_RADIUS + SIDEPLATE + 101.2 ); ! 101.2 Represents the middle between the sideplate and anchor lug
	SP_AGFY_E.trans.y := 13.5;!(yeager changed it 12-01-17)
	SP_AGFY_E.trans.z := -25 ;!(yeager changed it 12-01-17)

	SP_AGFY_S.trans.x := (FAMILY_GX.trans.x + NOZZLE_RADIUS + SIDEPLATE + 101.2 );
	SP_AGFY_S.trans.y := 48.5 ;!(yeager changed it 12-01-17)
	SP_AGFY_S.trans.z := -25;!(yeager changed it 12-01-17)

	SP_AHFY_E.trans.x := (FAMILY_HX.trans.x - NOZZLE_RADIUS - SIDEPLATE - 101.2 ); ! 101.2 Represents the middle between the sideplate and anchor lug
	SP_AHFY_E.trans.y := 13.5;!(yeager changed it 12-01-17)
	SP_AHFY_E.trans.z := -25 ;!(yeager changed it 12-01-17)

	SP_AHFY_S.trans.x := (FAMILY_HX.trans.x - NOZZLE_RADIUS - SIDEPLATE - 101.2 );
	SP_AHFY_S.trans.y := 48.5  ;!(yeager changed it 12-01-17)
	SP_AHFY_S.trans.z := -25 ;!(yeager changed it 12-01-17)

ENDIF


    ELSE IF ANCHOR_USED = 6802707 THEN

    IF WOTOX < 1500 THEN
     ! for short wotox!

	! ANCHOR "Y TOP" SEARCH  L & R
	SP_AGBY_E.trans.x := (FAMILY_GX.trans.x + NOZZLE_RADIUS + SIDEPLATE + 60.5 ); ! 72.5 Represents the distance from the sideplate to the center of the anchor lug
	SP_AGBY_E.trans.y := -13.5;	! Yeager changed this 12-27-17!
	SP_AGBY_E.trans.z := -125;	! Yeager changed this 12-27-17!

	SP_AGBY_S.trans.x := (FAMILY_GX.trans.x + NOZZLE_RADIUS + SIDEPLATE + 60.5 );  ! 72.5 Represents the distance from the sideplate to the center of the anchor lug
	SP_AGBY_S.trans.y := -43.5;	! Yeager changed this 12-27-17!
	SP_AGBY_S.trans.z := -125;	! Yeager changed this 12-27-17!

    SP_AHBY_E.trans.x := (FAMILY_HX.trans.x - NOZZLE_RADIUS - SIDEPLATE - 60.5 ); !72.5 Represents the distance from the sideplate to the center of the anchor lug
	SP_AHBY_E.trans.y := -13.5; ! Yeager changed this 12-27-17! on the casing
	SP_AHBY_E.trans.z := -125;	! Yeager changed this 12-27-17!

	SP_AHBY_S.trans.x := (FAMILY_HX.trans.x - NOZZLE_RADIUS - SIDEPLATE - 60.5 );  ! 72.5 Represents the distance from the sideplate to the center of the anchor lug
	SP_AHBY_S.trans.y := -43.5;	! Yeager changed this 12-27-17!
	SP_AHBY_S.trans.z := -125;	! Yeager changed this 12-27-17!
    ELSE
	! ANCHOR "Y TOP" SEARCH  L & R
	SP_AGBY_E.trans.x := (FAMILY_GX.trans.x + NOZZLE_RADIUS + SIDEPLATE + 60.5 ); ! 72.5 Represents the distance from the sideplate to the center of the anchor lug
	SP_AGBY_E.trans.y := 0;		! NOZZLE_RADIUS REPRESENTS the nozzle flush on the casing
	SP_AGBY_E.trans.z := -50 ;		! Represents distance from lug tangent to anchor body

	SP_AGBY_S.trans.x := (FAMILY_GX.trans.x + NOZZLE_RADIUS + SIDEPLATE + 60.5 );  ! 72.5 Represents the distance from the sideplate to the center of the anchor lug
	SP_AGBY_S.trans.y := -30;		! NOZZLE_RADIUS REPRESENTS the nozzle flush on the casing
	SP_AGBY_S.trans.z := -50 ;		! Represents distance from lug tangent to anchor body

    SP_AHBY_E.trans.x := (FAMILY_HX.trans.x - NOZZLE_RADIUS - SIDEPLATE - 60.5 ); !72.5 Represents the distance from the sideplate to the center of the anchor lug
	SP_AHBY_E.trans.y := 0;	! NOZZLE_RADIUS REPRESENTS the nozzle flush on the casing
	SP_AHBY_E.trans.z := -50 ;	! Represents distance from lug tangent to anchor body

	SP_AHBY_S.trans.x := (FAMILY_HX.trans.x - NOZZLE_RADIUS - SIDEPLATE - 60.5 );  ! 72.5 Represents the distance from the sideplate to the center of the anchor lug
	SP_AHBY_S.trans.y := -30;		! NOZZLE_RADIUS REPRESENTS the nozzle flush on the casing
	SP_AHBY_S.trans.z := -50 ;		! Represents distance from lug tangent to anchor body
  ENDIF
	    ! ANCHOR "Z TOP" SEARCH L & R
	SP_AGBZ_E.trans.x := (FAMILY_GX.trans.x + NOZZLE_RADIUS + SIDEPLATE + 60.5 ); ! 72.5 Represents the distance from the sideplate to the center of the anchor lug
	SP_AGBZ_E.trans.y := 75;    ! Represents roughly the wire STICK_OUT (TCP) to be below the flat bottom of the anchor
	SP_AGBZ_E.trans.z := NOZZLE_RADIUS;

	SP_AGBZ_S.trans.x := (FAMILY_GX.trans.x + NOZZLE_RADIUS + SIDEPLATE + 60.5 ); ! 72.5 Represents the distance from the sideplate to the center of the anchor lug
	SP_AGBZ_S.trans.y := 75;     ! Represents roughly the wire STICK_OUT (TCP) to be below the flat bottom of the anchor
	SP_AGBZ_S.trans.z := NOZZLE_RADIUS + 30;	!!  just a search length

	SP_AHBZ_E.trans.x := (FAMILY_HX.trans.x - NOZZLE_RADIUS - SIDEPLATE - 60.5 ); ! 72.5 Represents the distance from the sideplate to the center of the anchor lug
	SP_AHBZ_E.trans.y := 75;	! Represents roughly the wire STICK_OUT (TCP) to be below the flat bottom of the anchor
	SP_AHBZ_E.trans.z := NOZZLE_RADIUS;

	SP_AHBZ_S.trans.x := (FAMILY_HX.trans.x - NOZZLE_RADIUS - SIDEPLATE - 60.5 ); ! 72.5 Represents the distance from the sideplate to the center of the anchor lug
	SP_AHBZ_S.trans.y := 75;	! Represents roughly the wire STICK_OUT (TCP) to be below the flat bottom of the anchor
	SP_AHBZ_S.trans.z := NOZZLE_RADIUS + 30; !!  just a search length


    IF WOTOX < 1500 THEN
     ! for short wotox!
	! ANCHOR "Y BOTTOM" SEARCH  L & R
	SP_AGFY_E.trans.x := (FAMILY_GX.trans.x + NOZZLE_RADIUS + SIDEPLATE + 60.5 ); ! 72.5 Represents the distance from the sideplate to the center of the anchor lug
	SP_AGFY_E.trans.y := 13.5;	! Yeager changed this 12-27-17!
	SP_AGFY_E.trans.z := -125 ;! Yeager changed this 12-27-17!

	SP_AGFY_S.trans.x := (FAMILY_GX.trans.x + NOZZLE_RADIUS + SIDEPLATE + 60.5 );  ! 72.5 Represents the distance from the sideplate to the center of the anchor lug
	SP_AGFY_S.trans.y := 43.5;! Yeager changed this 12-27-17!
	SP_AGFY_S.trans.z := -125 ;! Yeager changed this 12-27-17!

    SP_AHFY_E.trans.x := (FAMILY_HX.trans.x - NOZZLE_RADIUS - SIDEPLATE - 60.5 ); !72.5 Represents the distance from the sideplate to the center of the anchor lug
	SP_AHFY_E.trans.y := 13.5;	! Yeager changed this 12-27-17!
	SP_AHFY_E.trans.z := -125 ;! Yeager changed this 12-27-17!

	SP_AHFY_S.trans.x := (FAMILY_HX.trans.x - NOZZLE_RADIUS - SIDEPLATE - 60.5 );  ! 72.5 Represents the distance from the sideplate to the center of the anchor lug
	SP_AHFY_S.trans.y := 43.5;! Yeager changed this 12-27-17!
	SP_AHFY_S.trans.z := -125 ;! Yeager changed this 12-27-17!
	ELSE
	! ANCHOR "Y BOTTOM" SEARCH  L & R
	SP_AGFY_E.trans.x := (FAMILY_GX.trans.x + NOZZLE_RADIUS + SIDEPLATE + 60.5 ); ! 72.5 Represents the distance from the sideplate to the center of the anchor lug
	SP_AGFY_E.trans.y := 0;		! NOZZLE_RADIUS REPRESENTS the nozzle flush on the casting
	SP_AGFY_E.trans.z := -40 ;		! Represents distance from lug tangent to anchor body

	SP_AGFY_S.trans.x := (FAMILY_GX.trans.x + NOZZLE_RADIUS + SIDEPLATE + 60.5 );  ! 72.5 Represents the distance from the sideplate to the center of the anchor lug
	SP_AGFY_S.trans.y := 25;		! NOZZLE_RADIUS REPRESENTS the nozzle flush on the casting
	SP_AGFY_S.trans.z := -40 ;		! Represents distance from lug tangent to anchor body

    SP_AHFY_E.trans.x := (FAMILY_HX.trans.x - NOZZLE_RADIUS - SIDEPLATE - 60.5 ); !72.5 Represents the distance from the sideplate to the center of the anchor lug
	SP_AHFY_E.trans.y := 0;	! NOZZLE_RADIUS REPRESENTS the nozzle flush on the casing
	SP_AHFY_E.trans.z := -40 ;	! Represents distance from lug tangent to anchor body

	SP_AHFY_S.trans.x := (FAMILY_HX.trans.x - NOZZLE_RADIUS - SIDEPLATE - 60.5 );  ! 72.5 Represents the distance from the sideplate to the center of the anchor lug
	SP_AHFY_S.trans.y := 25;		! NOZZLE_RADIUS REPRESENTS the nozzle flush on the casting
	SP_AHFY_S.trans.z := -40 ;		! Represents distance from lug tangent to anchor body

  ENDIF
	! ANCHOR "Z BOTTOM" SEARCH L & R

    SP_AGFZ_E.trans.x := (FAMILY_GX.trans.x + NOZZLE_RADIUS + SIDEPLATE + 60.5 ); ! 72.5 Represents the distance from the sideplate to the center of the anchor lug
	SP_AGFZ_E.trans.y := -90;    ! Represents roughly the wire STICK_OUT (TCP) to be below the flat bottom of the anchor
	SP_AGFZ_E.trans.z := NOZZLE_RADIUS;

	SP_AGFZ_S.trans.x := (FAMILY_GX.trans.x + NOZZLE_RADIUS + SIDEPLATE + 60.5 ); ! 72.5 Represents the distance from the sideplate to the center of the anchor lug
	SP_AGFZ_S.trans.y := -90;     ! Represents roughly the wire STICK_OUT (TCP) to be below the flat bottom of the anchor
	SP_AGFZ_S.trans.z := NOZZLE_RADIUS + 30;	!!  just a search length

	SP_AHFZ_E.trans.x := (FAMILY_HX.trans.x - NOZZLE_RADIUS - SIDEPLATE - 60.5 ); ! 72.5 Represents the distance from the sideplate to the center of the anchor lug
	SP_AHFZ_E.trans.y := -90;	! Represents roughly the wire STICK_OUT (TCP) to be below the flat bottom of the anchor
	SP_AHFZ_E.trans.z := NOZZLE_RADIUS;

	SP_AHFZ_S.trans.x := (FAMILY_HX.trans.x - NOZZLE_RADIUS - SIDEPLATE - 60.5 ); ! 72.5 Represents the distance from the sideplate to the center of the anchor lug
	SP_AHFZ_S.trans.y := -90;	! Represents roughly the wire STICK_OUT (TCP) to be below the flat bottom of the anchor
	SP_AHFZ_S.trans.z := NOZZLE_RADIUS + 30; !!  just a search length

	! ANCHOR BACK "X" SEARCH G & H

	SP_GX_E.trans.x := (FAMILY_GX.trans.x + (NOZZLE_RADIUS*2) + SIDEPLATE  );
	SP_GX_E.trans.y := 0;
	SP_GX_E.trans.z := 30;  ! distance behind the lug of the anchor

	SP_GX_S.trans.x := (FAMILY_GX.trans.x + (NOZZLE_RADIUS*2) + SIDEPLATE + 25 ); ! 30 Represents generic search length
	SP_GX_S.trans.y := 0;
	SP_GX_S.trans.z := 30;	! distance behind the lug of the anchor

	SP_HX_E.trans.x := (FAMILY_HX.trans.x - (NOZZLE_RADIUS*2) - SIDEPLATE  );
	SP_HX_E.trans.y := 0;
	SP_HX_E.trans.z := 30;	! distance behind the lug of the anchor

	SP_HX_S.trans.x := (FAMILY_HX.trans.x - (NOZZLE_RADIUS*2) - SIDEPLATE - 25 ); ! 30 Represents generic search length
	SP_HX_S.trans.y := 0;
	SP_HX_S.trans.z := 30;		! distance behind the lug of the anchor


        ! ANCHOR FRONT  "X" SEARCH G & H
	SP_AGFX_E.trans.x := FAMILY_GX.trans.x  + SIDEPLATE + (2 * NOZZLE_RADIUS); ! 40 Represents Search Distance
	SP_AGFX_E.trans.y := -50;
	SP_AGFX_E.trans.z := NOZZLE_RADIUS + 30;

	SP_AGFX_S.trans.x := FAMILY_GX.trans.x  + SIDEPLATE + (2 * NOZZLE_RADIUS) + 40;
	SP_AGFX_S.trans.y := -50;
	SP_AGFX_S.trans.z := NOZZLE_RADIUS + 30;

!!!!!!!!!!!!!!!!!!!!!!!!!!!!!!!!!!!!!!!!!!!!
	SP_AHFX_E.trans.x := FAMILY_HX.trans.x - SIDEPLATE - (2 * NOZZLE_RADIUS); ! 40 Represents Search Distance
	SP_AHFX_E.trans.y := -50;
	SP_AHFX_E.trans.z := NOZZLE_RADIUS + 30;

	SP_AHFX_S.trans.x := FAMILY_HX.trans.x - SIDEPLATE - (2 * NOZZLE_RADIUS) - 40;
	SP_AHFX_S.trans.y := -50;
	SP_AHFX_S.trans.z := NOZZLE_RADIUS + 30;


ELSEIF ANCHOR_USED = 689899 THEN

	! ANCHOR "Y BACK" SEARCH  L & R
	SP_AGBY_E.trans.x := (FAMILY_GX.trans.x + NOZZLE_RADIUS + SIDEPLATE + 88.5 ); ! 44 Represents the middle between the sideplate and anchor lug
	SP_AGBY_E.trans.y := 0;
	SP_AGBY_E.trans.z := -102.5 ;

	SP_AGBY_S.trans.x := (FAMILY_GX.trans.x + NOZZLE_RADIUS + SIDEPLATE + 88.5 );
	SP_AGBY_S.trans.y := -30;
	SP_AGBY_S.trans.z := -102.5 ;

	SP_AHBY_E.trans.x := (FAMILY_HX.trans.x - NOZZLE_RADIUS - SIDEPLATE - 88.5 ); ! 44 Represents the middle between the sideplate and anchor lug
	SP_AHBY_E.trans.y := 0;
	SP_AHBY_E.trans.z := -102.5;

	SP_AHBY_S.trans.x := (FAMILY_HX.trans.x - NOZZLE_RADIUS - SIDEPLATE - 88.5);
	SP_AHBY_S.trans.y := -30;
	SP_AHBY_S.trans.z := -102.5 ;

  	! ANCHOR "Y FRONT" SEARCH  L & R
	SP_AGFY_E.trans.x := (FAMILY_GX.trans.x + NOZZLE_RADIUS + SIDEPLATE + 83.5 ); ! 44 Represents the middle between the sideplate and anchor lug
	SP_AGFY_E.trans.y := 0;
	SP_AGFY_E.trans.z := -102.5 ;

	SP_AGFY_S.trans.x := (FAMILY_GX.trans.x + NOZZLE_RADIUS + SIDEPLATE + 83.5 );
	SP_AGFY_S.trans.y := 25  ;
	SP_AGFY_S.trans.z := -102.5 ;

	SP_AHFY_E.trans.x := (FAMILY_HX.trans.x - NOZZLE_RADIUS - SIDEPLATE - 83.5 ); ! 44 Represents the middle between the sideplate and anchor lug
	SP_AHFY_E.trans.y := 0;
	SP_AHFY_E.trans.z := -102.5 ;

	SP_AHFY_S.trans.x := (FAMILY_HX.trans.x - NOZZLE_RADIUS - SIDEPLATE - 83.5 );
	SP_AHFY_S.trans.y := 25;
	SP_AHFY_S.trans.z := -102.5 ;

    ! ANCHOR BACK  "Z" SEARCH L & R
	SP_AGBZ_E.trans.x := (FAMILY_GX.trans.x + NOZZLE_RADIUS + SIDEPLATE + 83.4 ); ! 102.5 Represents distance from the sideplate to the center of the Anchor lug
	SP_AGBZ_E.trans.y := 60;
	SP_AGBZ_E.trans.z := NOZZLE_RADIUS;

	SP_AGBZ_S.trans.x := (FAMILY_GX.trans.x + NOZZLE_RADIUS + SIDEPLATE + 83.4 );
	SP_AGBZ_S.trans.y := 60;
	SP_AGBZ_S.trans.z := NOZZLE_RADIUS + 30;

	SP_AHBZ_E.trans.x := (FAMILY_HX.trans.x - NOZZLE_RADIUS - SIDEPLATE - 83.4 ); ! 102.5 Represents distance from the sideplate to the center of the Anchor lug
	SP_AHBZ_E.trans.y := 60;
	SP_AHBZ_E.trans.z := NOZZLE_RADIUS;

	SP_AHBZ_S.trans.x := (FAMILY_HX.trans.x - NOZZLE_RADIUS - SIDEPLATE - 83.4 );
	SP_AHBZ_S.trans.y := 60;
	SP_AHBZ_S.trans.z := NOZZLE_RADIUS + 30;

        ! ANCHOR FRONT  "Z" SEARCH L & R
	SP_AGFZ_E.trans.x := (FAMILY_GX.trans.x + NOZZLE_RADIUS + SIDEPLATE + 83.4 ); ! 102.5 Represents distance from the sideplate to the center of the Anchor lug
	SP_AGFZ_E.trans.y := -75;
	SP_AGFZ_E.trans.z := NOZZLE_RADIUS;

	SP_AGFZ_S.trans.x := (FAMILY_GX.trans.x + NOZZLE_RADIUS + SIDEPLATE + 83.4 );
	SP_AGFZ_S.trans.y := -75;
	SP_AGFZ_S.trans.z := NOZZLE_RADIUS + 30;

	SP_AHFZ_E.trans.x := (FAMILY_HX.trans.x - NOZZLE_RADIUS - SIDEPLATE - 83.4 ); ! 102.5 Represents distance from the sideplate to the center of the Anchor lug
	SP_AHFZ_E.trans.y := -75;
	SP_AHFZ_E.trans.z := NOZZLE_RADIUS;

	SP_AHFZ_S.trans.x := (FAMILY_HX.trans.x - NOZZLE_RADIUS - SIDEPLATE - 83.4 );
	SP_AHFZ_S.trans.y := -75;
	SP_AHFZ_S.trans.z := NOZZLE_RADIUS + 30;

    ! ANCHOR BACK "X" SEARCH G & H

	SP_GX_E.trans.x := (FAMILY_GX.trans.x + (NOZZLE_RADIUS*2) + SIDEPLATE  );
	SP_GX_E.trans.y := 0;
	SP_GX_E.trans.z := 35;

	SP_GX_S.trans.x := (FAMILY_GX.trans.x + (NOZZLE_RADIUS*2) + SIDEPLATE + 30 ); !30 Represents generic search length
	SP_GX_S.trans.y := 0;
	SP_GX_S.trans.z := 35;

	SP_HX_E.trans.x := (FAMILY_HX.trans.x - (NOZZLE_RADIUS*2) - SIDEPLATE  );
	SP_HX_E.trans.y := 0;
	SP_HX_E.trans.z := 35;

	SP_HX_S.trans.x := (FAMILY_HX.trans.x - (NOZZLE_RADIUS*2) - SIDEPLATE - 30 ); !30 Represents generic search length
	SP_HX_S.trans.y := 0;
	SP_HX_S.trans.z := 35;


        ! ANCHOR FRONT  "X" SEARCH G & H
	SP_AGFX_E.trans.x := FAMILY_GX.trans.x  + SIDEPLATE + (2 * NOZZLE_RADIUS); ! 40 Represents Search Distance
	SP_AGFX_E.trans.y := -50;
	SP_AGFX_E.trans.z := NOZZLE_RADIUS + 30;

	SP_AGFX_S.trans.x := FAMILY_GX.trans.x  + SIDEPLATE + (2 * NOZZLE_RADIUS) + 40;
	SP_AGFX_S.trans.y := -50;
	SP_AGFX_S.trans.z := NOZZLE_RADIUS + 30;

!!!!!!!!!!!!!!!!!!!!!!!!!!!!!!!!!!!!!!!!!!!!
	SP_AHFX_E.trans.x := FAMILY_HX.trans.x - SIDEPLATE - (2 * NOZZLE_RADIUS); ! 40 Represents Search Distance
	SP_AHFX_E.trans.y := -50;
	SP_AHFX_E.trans.z := NOZZLE_RADIUS + 30;

	SP_AHFX_S.trans.x := FAMILY_HX.trans.x - SIDEPLATE - (2 * NOZZLE_RADIUS) - 40;
	SP_AHFX_S.trans.y := -50;
	SP_AHFX_S.trans.z := NOZZLE_RADIUS + 30;


ELSEIF ANCHOR_USED = 6862141 THEN
	! ANCHOR "Y BACK" SEARCH  L & R
	SP_AGBY_E.trans.x := (FAMILY_GX.trans.x + NOZZLE_RADIUS + SIDEPLATE + 65.5 ); !Yeager changed on 12-05-17
	SP_AGBY_E.trans.y := -13.5; !Yeager changed on 12-05-17
	SP_AGBY_E.trans.z := -65 ; !Yeager changed on 12-05-17

	SP_AGBY_S.trans.x := (FAMILY_GX.trans.x + NOZZLE_RADIUS + SIDEPLATE + 65.5 ); !Yeager changed on 12-05-17
	SP_AGBY_S.trans.y := -53.5 ; !Yeager changed on 12-05-17
	SP_AGBY_S.trans.z := -65 ; !Yeager changed on 12-05-17

	SP_AHBY_E.trans.x := (FAMILY_HX.trans.x - NOZZLE_RADIUS - SIDEPLATE - 65.5 ); !Yeager changed on 12-05-17
	SP_AHBY_E.trans.y := -13.5; !Yeager changed on 12-05-17
	SP_AHBY_E.trans.z := -65 ; !Yeager changed on 12-05-17

	SP_AHBY_S.trans.x := (FAMILY_HX.trans.x - NOZZLE_RADIUS - SIDEPLATE - 65.5 ); !Yeager changed on 12-05-17
	SP_AHBY_S.trans.y := -53.5 ;!Yeager changed on 12-05-17
	SP_AHBY_S.trans.z := -65 ; !Yeager changed on 12-05-17

    IF WOTOX < 1400 THEN
     ! for short wotox!

   	! ANCHOR "Y FRONT" SEARCH  L & R
	SP_AGFY_E.trans.x := (FAMILY_GX.trans.x + NOZZLE_RADIUS + SIDEPLATE + 76.5 ); !Yeager changed on 12-05-17
	SP_AGFY_E.trans.y := 13.5;	!Yeager changed on 01-21-18
	SP_AGFY_E.trans.z := -125 ;	!Yeager changed on 01-21-18

	SP_AGFY_S.trans.x := (FAMILY_GX.trans.x + NOZZLE_RADIUS + SIDEPLATE + 76.5 ); !Yeager changed on 12-05-17
	SP_AGFY_S.trans.y := 53.5; !Yeager changed on 01-21-18
	SP_AGFY_S.trans.z := -125; !Yeager changed on 01-21-18

	SP_AHFY_E.trans.x := (FAMILY_HX.trans.x - NOZZLE_RADIUS - SIDEPLATE - 76.5 ); !Yeager changed on 12-05-17
	SP_AHFY_E.trans.y := 13.5; !Yeager changed on 01-21-18
	SP_AHFY_E.trans.z := -125; !Yeager changed on 01-21-18

	SP_AHFY_S.trans.x := (FAMILY_HX.trans.x - NOZZLE_RADIUS - SIDEPLATE - 76.5 ); !Yeager changed on 12-05-17
	SP_AHFY_S.trans.y := 53.5; !Yeager changed on 01-21-18
	SP_AHFY_S.trans.z := -125; !Yeager changed on 01-21-18

    ELSE


  	! ANCHOR "Y FRONT" SEARCH  L & R
	SP_AGFY_E.trans.x := (FAMILY_GX.trans.x + NOZZLE_RADIUS + SIDEPLATE + 76.5 ); !Yeager changed on 12-05-17
	SP_AGFY_E.trans.y := 13.5;
	SP_AGFY_E.trans.z := 10 ;

	SP_AGFY_S.trans.x := (FAMILY_GX.trans.x + NOZZLE_RADIUS + SIDEPLATE + 76.5 ); !Yeager changed on 12-05-17
	SP_AGFY_S.trans.y := 53.5; !Yeager changed on 12-05-17
	SP_AGFY_S.trans.z := 10; !Yeager changed on 12-05-17

	SP_AHFY_E.trans.x := (FAMILY_HX.trans.x - NOZZLE_RADIUS - SIDEPLATE - 76.5 ); !Yeager changed on 12-05-17
	SP_AHFY_E.trans.y := 13.5; !Yeager changed on 12-05-17
	SP_AHFY_E.trans.z := 10; !Yeager changed on 12-05-17

	SP_AHFY_S.trans.x := (FAMILY_HX.trans.x - NOZZLE_RADIUS - SIDEPLATE - 76.5 ); !Yeager changed on 12-05-17
	SP_AHFY_S.trans.y := 53.5; !Yeager changed on 12-05-17
	SP_AHFY_S.trans.z := 10; !Yeager changed on 12-05-17
    ENDIF
    ! ANCHOR BACK  "Z" SEARCH L & R
	SP_AGBZ_E.trans.x := (FAMILY_GX.trans.x + NOZZLE_RADIUS + SIDEPLATE + 76.5 ); ! 102.5 Represents distance from the sideplate to the center of the Anchor lug
	SP_AGBZ_E.trans.y := 75;
	SP_AGBZ_E.trans.z := NOZZLE_RADIUS;

	SP_AGBZ_S.trans.x := (FAMILY_GX.trans.x + NOZZLE_RADIUS + SIDEPLATE + 76.5 );
	SP_AGBZ_S.trans.y := 75;
	SP_AGBZ_S.trans.z := NOZZLE_RADIUS + 30;

	SP_AHBZ_E.trans.x := (FAMILY_HX.trans.x - NOZZLE_RADIUS - SIDEPLATE - 76.5); ! 102.5 Represents distance from the sideplate to the center of the Anchor lug
	SP_AHBZ_E.trans.y := 75;
	SP_AHBZ_E.trans.z := NOZZLE_RADIUS;

	SP_AHBZ_S.trans.x := (FAMILY_HX.trans.x - NOZZLE_RADIUS - SIDEPLATE - 76.5 );
	SP_AHBZ_S.trans.y := 75;
	SP_AHBZ_S.trans.z := NOZZLE_RADIUS + 30;

        ! ANCHOR FRONT  "Z" SEARCH L & R
	SP_AGFZ_E.trans.x := (FAMILY_GX.trans.x + NOZZLE_RADIUS + SIDEPLATE + 76.5 ); ! 102.5 Represents distance from the sideplate to the center of the Anchor lug
	SP_AGFZ_E.trans.y := -95; !Yeager changed on 12-05-17
	SP_AGFZ_E.trans.z := NOZZLE_RADIUS;

	SP_AGFZ_S.trans.x := (FAMILY_GX.trans.x + NOZZLE_RADIUS + SIDEPLATE + 76.5 );
	SP_AGFZ_S.trans.y := -95; !Yeager changed on 12-05-17
	SP_AGFZ_S.trans.z := NOZZLE_RADIUS + 30;

	SP_AHFZ_E.trans.x := (FAMILY_HX.trans.x - NOZZLE_RADIUS - SIDEPLATE - 76.5 ); ! 102.5 Represents distance from the sideplate to the center of the Anchor lug
	SP_AHFZ_E.trans.y := -95; !Yeager changed on 12-05-17
	SP_AHFZ_E.trans.z := NOZZLE_RADIUS;

	SP_AHFZ_S.trans.x := (FAMILY_HX.trans.x - NOZZLE_RADIUS - SIDEPLATE - 76.5 );
	SP_AHFZ_S.trans.y := -95; !Yeager changed on 12-05-17
	SP_AHFZ_S.trans.z := NOZZLE_RADIUS + 30;

    ! ANCHOR BACK "X" SEARCH G & H

	SP_GX_E.trans.x := (FAMILY_GX.trans.x + (NOZZLE_RADIUS*2) + SIDEPLATE  );
	SP_GX_E.trans.y := 0;
	SP_GX_E.trans.z := 65;

	SP_GX_S.trans.x := (FAMILY_GX.trans.x + (NOZZLE_RADIUS*2) + SIDEPLATE + 30 ); !30 Represents generic search length
	SP_GX_S.trans.y := 0;
	SP_GX_S.trans.z := 65;

	SP_HX_E.trans.x := (FAMILY_HX.trans.x - (NOZZLE_RADIUS*2) - SIDEPLATE  );
	SP_HX_E.trans.y := 0;
	SP_HX_E.trans.z := 65;

	SP_HX_S.trans.x := (FAMILY_HX.trans.x - (NOZZLE_RADIUS*2) - SIDEPLATE - 30 ); !30 Represents generic search length
	SP_HX_S.trans.y := 0;
	SP_HX_S.trans.z := 65;

        ! ANCHOR FRONT  "X" SEARCH G & H
	SP_AGFX_E.trans.x := FAMILY_GX.trans.x  + SIDEPLATE + (2 * NOZZLE_RADIUS); ! 40 Represents Search Distance
	SP_AGFX_E.trans.y := -50;
	SP_AGFX_E.trans.z := NOZZLE_RADIUS + 30;

	SP_AGFX_S.trans.x := FAMILY_GX.trans.x  + SIDEPLATE + (2 * NOZZLE_RADIUS) + 40;
	SP_AGFX_S.trans.y := -50;
	SP_AGFX_S.trans.z := NOZZLE_RADIUS + 30;

!!!!!!!!!!!!!!!!!!!!!!!!!!!!!!!!!!!!!!!!!!!!
	SP_AHFX_E.trans.x := FAMILY_HX.trans.x - SIDEPLATE - (2 * NOZZLE_RADIUS); ! 40 Represents Search Distance
	SP_AHFX_E.trans.y := -50;
	SP_AHFX_E.trans.z := NOZZLE_RADIUS + 30;

	SP_AHFX_S.trans.x := FAMILY_HX.trans.x - SIDEPLATE - (2 * NOZZLE_RADIUS) - 40;
	SP_AHFX_S.trans.y := -50;
	SP_AHFX_S.trans.z := NOZZLE_RADIUS + 30;

ENDIF
ENDIF
ENDIF
ENDIF
ENDIF

HOPE_IT_WORKS:

    ENDPROC

    PROC SET_ANCHOR_X(INOUT
   ROBTARGET FRONT_OR_BACK_X_FOUND)
!!!!!!!!!!!!!!!!REVISED 03-16-18 to add anchor_back X searches!!!!!
	PDispOff;
    IF  FRONT_OR_BACK_X_FOUND.trans.x > 0 THEN
!!!!!!!!!!!!!!!!!!!!!!!!!!!!!!!!!!!!!!!!!!!!!!!!!!!!!!!!!!!!!!!!!!!!!!!!!
!                 ALL H SIDE ANCHOR X VALUES FOR SQUARE ANCHORS
   	AH200.trans.x := (FRONT_OR_BACK_X_FOUND.trans.x + NOZZLE_RADIUS) - STICK_OUT;
    AH201.trans.x := (FRONT_OR_BACK_X_FOUND.trans.x + NOZZLE_RADIUS) - STICK_OUT;
   	AH202.trans.x := (FRONT_OR_BACK_X_FOUND.trans.x + NOZZLE_RADIUS) - STICK_OUT;
    AH203.trans.x := (FRONT_OR_BACK_X_FOUND.trans.x + NOZZLE_RADIUS) - STICK_OUT;
  	AH204.trans.x := (FRONT_OR_BACK_X_FOUND.trans.x + NOZZLE_RADIUS) - STICK_OUT;
  	AH205.trans.x := (FRONT_OR_BACK_X_FOUND.trans.x + NOZZLE_RADIUS) - STICK_OUT;
  	AH206.trans.x := (FRONT_OR_BACK_X_FOUND.trans.x + NOZZLE_RADIUS) - STICK_OUT;
  	AH207.trans.x := (FRONT_OR_BACK_X_FOUND.trans.x + NOZZLE_RADIUS) - STICK_OUT;
  	AH208.trans.x := (FRONT_OR_BACK_X_FOUND.trans.x + NOZZLE_RADIUS) - STICK_OUT;
   	AH209.trans.x := (FRONT_OR_BACK_X_FOUND.trans.x + NOZZLE_RADIUS) - STICK_OUT;
  	AH210.trans.x := (FRONT_OR_BACK_X_FOUND.trans.x + NOZZLE_RADIUS) - STICK_OUT;
  	AH218.trans.x := (FRONT_OR_BACK_X_FOUND.trans.x + NOZZLE_RADIUS) - STICK_OUT;
  	AH219.trans.x := (FRONT_OR_BACK_X_FOUND.trans.x + NOZZLE_RADIUS) - STICK_OUT;
  	AH220.trans.x := (FRONT_OR_BACK_X_FOUND.trans.x + NOZZLE_RADIUS) - STICK_OUT;
!!!!!!!!!!!!!!!!!!!!!!!!!!!!!!!!!!!!!!!!!!!!!!!!!!!!!!!!!!!!!!!!!!!!!!!!!

!                 ALL H SIDE ANCHOR X VALUES  FOR "H" ANCHORS
   	AH300.trans.x := (FRONT_OR_BACK_X_FOUND.trans.x + NOZZLE_RADIUS) - STICK_OUT;
    AH301.trans.x := (FRONT_OR_BACK_X_FOUND.trans.x + NOZZLE_RADIUS) - STICK_OUT;
   	AH302.trans.x := (FRONT_OR_BACK_X_FOUND.trans.x + NOZZLE_RADIUS) - STICK_OUT;
    AH303.trans.x := (FRONT_OR_BACK_X_FOUND.trans.x + NOZZLE_RADIUS) - STICK_OUT;
  	AH304.trans.x := (FRONT_OR_BACK_X_FOUND.trans.x + NOZZLE_RADIUS) - STICK_OUT;
  	AH306.trans.x := (FRONT_OR_BACK_X_FOUND.trans.x + NOZZLE_RADIUS) - STICK_OUT;
  	AH307.trans.x := (FRONT_OR_BACK_X_FOUND.trans.x + NOZZLE_RADIUS) - STICK_OUT;
  	AH308.trans.x := (FRONT_OR_BACK_X_FOUND.trans.x + NOZZLE_RADIUS) - STICK_OUT;
   	AH309.trans.x := (FRONT_OR_BACK_X_FOUND.trans.x + NOZZLE_RADIUS) - STICK_OUT;
  	AH310.trans.x := (FRONT_OR_BACK_X_FOUND.trans.x + NOZZLE_RADIUS) - STICK_OUT;

    !                 ALL H SIDE ANCHOR X VALUES FOR SQUARE ANCHORS
   	AH400.trans.x := (FRONT_OR_BACK_X_FOUND.trans.x + NOZZLE_RADIUS) - STICK_OUT;
    AH401.trans.x := (FRONT_OR_BACK_X_FOUND.trans.x + NOZZLE_RADIUS) - STICK_OUT;
   	AH402.trans.x := (FRONT_OR_BACK_X_FOUND.trans.x + NOZZLE_RADIUS) - STICK_OUT;
    AH403.trans.x := (FRONT_OR_BACK_X_FOUND.trans.x + NOZZLE_RADIUS) - STICK_OUT;
  	AH404.trans.x := (FRONT_OR_BACK_X_FOUND.trans.x + NOZZLE_RADIUS) - STICK_OUT;
  	AH405.trans.x := (FRONT_OR_BACK_X_FOUND.trans.x + NOZZLE_RADIUS) - STICK_OUT;
  	AH406.trans.x := (FRONT_OR_BACK_X_FOUND.trans.x + NOZZLE_RADIUS) - STICK_OUT;
  	AH407.trans.x := (FRONT_OR_BACK_X_FOUND.trans.x + NOZZLE_RADIUS) - STICK_OUT;
  	AH408.trans.x := (FRONT_OR_BACK_X_FOUND.trans.x + NOZZLE_RADIUS) - STICK_OUT;
   	AH409.trans.x := (FRONT_OR_BACK_X_FOUND.trans.x + NOZZLE_RADIUS) - STICK_OUT;
  	AH410.trans.x := (FRONT_OR_BACK_X_FOUND.trans.x + NOZZLE_RADIUS) - STICK_OUT;
  	AH418.trans.x := (FRONT_OR_BACK_X_FOUND.trans.x + NOZZLE_RADIUS) - STICK_OUT;
  	AH419.trans.x := (FRONT_OR_BACK_X_FOUND.trans.x + NOZZLE_RADIUS) - STICK_OUT;
  	AH420.trans.x := (FRONT_OR_BACK_X_FOUND.trans.x + NOZZLE_RADIUS) - STICK_OUT;
    WaitTime\InPos, 0.5;


ELSEIF FRONT_OR_BACK_X_FOUND.trans.x < 0 THEN

!                 ALL G SIDE ANCHOR X VALUES FOR SQUARE ANCHORS
  	AG200.trans.x := (FRONT_OR_BACK_X_FOUND.trans.x - NOZZLE_RADIUS) + STICK_OUT;
    AG201.trans.x := (FRONT_OR_BACK_X_FOUND.trans.x - NOZZLE_RADIUS) + STICK_OUT;
    AG202.trans.x := (FRONT_OR_BACK_X_FOUND.trans.x - NOZZLE_RADIUS) + STICK_OUT;
  	AG203.trans.x := (FRONT_OR_BACK_X_FOUND.trans.x - NOZZLE_RADIUS) + STICK_OUT;
  	AG204.trans.x := (FRONT_OR_BACK_X_FOUND.trans.x - NOZZLE_RADIUS) + STICK_OUT;
    AG205.trans.x := (FRONT_OR_BACK_X_FOUND.trans.x - NOZZLE_RADIUS) + STICK_OUT;
  	AG206.trans.x := (FRONT_OR_BACK_X_FOUND.trans.x - NOZZLE_RADIUS) + STICK_OUT;
  	AG207.trans.x := (FRONT_OR_BACK_X_FOUND.trans.x - NOZZLE_RADIUS) + STICK_OUT;
  	AG208.trans.x := (FRONT_OR_BACK_X_FOUND.trans.x - NOZZLE_RADIUS) + STICK_OUT;
  	AG209.trans.x := (FRONT_OR_BACK_X_FOUND.trans.x - NOZZLE_RADIUS) + STICK_OUT;
  	AG210.trans.x := (FRONT_OR_BACK_X_FOUND.trans.x - NOZZLE_RADIUS) + STICK_OUT;
  	AG218.trans.x := (FRONT_OR_BACK_X_FOUND.trans.x - NOZZLE_RADIUS) + STICK_OUT;
  	AG219.trans.x := (FRONT_OR_BACK_X_FOUND.trans.x - NOZZLE_RADIUS) + STICK_OUT;
    AG220.trans.x := (FRONT_OR_BACK_X_FOUND.trans.x - NOZZLE_RADIUS) + STICK_OUT;

!!!!!!!!!!!!!!!!!!!!!!!!!!!!!!!!!!!!!!!!!!!!!!!!!!!!!!!!!!!!!!!!!!!!!!!!!
!                 ALL G SIDE ANCHOR X VALUES FOR "H" ANCHORS
  	AG300.trans.x := (FRONT_OR_BACK_X_FOUND.trans.x - NOZZLE_RADIUS) + STICK_OUT;
    AG301.trans.x := (FRONT_OR_BACK_X_FOUND.trans.x - NOZZLE_RADIUS) + STICK_OUT;
    AG302.trans.x := (FRONT_OR_BACK_X_FOUND.trans.x - NOZZLE_RADIUS) + STICK_OUT;
  	AG303.trans.x := (FRONT_OR_BACK_X_FOUND.trans.x - NOZZLE_RADIUS) + STICK_OUT;
  	AG304.trans.x := (FRONT_OR_BACK_X_FOUND.trans.x - NOZZLE_RADIUS) + STICK_OUT;
  	AG306.trans.x := (FRONT_OR_BACK_X_FOUND.trans.x - NOZZLE_RADIUS) + STICK_OUT;
  	AG307.trans.x := (FRONT_OR_BACK_X_FOUND.trans.x - NOZZLE_RADIUS) + STICK_OUT;
  	AG308.trans.x := (FRONT_OR_BACK_X_FOUND.trans.x - NOZZLE_RADIUS) + STICK_OUT;
  	AG309.trans.x := (FRONT_OR_BACK_X_FOUND.trans.x - NOZZLE_RADIUS) + STICK_OUT;
  	AG310.trans.x := (FRONT_OR_BACK_X_FOUND.trans.x - NOZZLE_RADIUS) + STICK_OUT;

!!!!!!!!!!!!!!!!!!!!!!!!!!!!!!!!!!!!!!!!!!!!!!!!!!!!!!!!!!!!!!!!!!!!!!!!!
!                 ALL G SIDE ANCHOR X VALUES FOR SQUARE ANCHORS
  	AG400.trans.x := (FRONT_OR_BACK_X_FOUND.trans.x - NOZZLE_RADIUS) + STICK_OUT;
    AG401.trans.x := (FRONT_OR_BACK_X_FOUND.trans.x - NOZZLE_RADIUS) + STICK_OUT;
    AG402.trans.x := (FRONT_OR_BACK_X_FOUND.trans.x - NOZZLE_RADIUS) + STICK_OUT;
  	AG403.trans.x := (FRONT_OR_BACK_X_FOUND.trans.x - NOZZLE_RADIUS) + STICK_OUT;
  	AG404.trans.x := (FRONT_OR_BACK_X_FOUND.trans.x - NOZZLE_RADIUS) + STICK_OUT;
    AG405.trans.x := (FRONT_OR_BACK_X_FOUND.trans.x - NOZZLE_RADIUS) + STICK_OUT;
  	AG406.trans.x := (FRONT_OR_BACK_X_FOUND.trans.x - NOZZLE_RADIUS) + STICK_OUT;
  	AG407.trans.x := (FRONT_OR_BACK_X_FOUND.trans.x - NOZZLE_RADIUS) + STICK_OUT;
  	AG408.trans.x := (FRONT_OR_BACK_X_FOUND.trans.x - NOZZLE_RADIUS) + STICK_OUT;
  	AG409.trans.x := (FRONT_OR_BACK_X_FOUND.trans.x - NOZZLE_RADIUS) + STICK_OUT;
  	AG410.trans.x := (FRONT_OR_BACK_X_FOUND.trans.x - NOZZLE_RADIUS) + STICK_OUT;
  	AG418.trans.x := (FRONT_OR_BACK_X_FOUND.trans.x - NOZZLE_RADIUS) + STICK_OUT;
  	AG419.trans.x := (FRONT_OR_BACK_X_FOUND.trans.x - NOZZLE_RADIUS) + STICK_OUT;
    AG420.trans.x := (FRONT_OR_BACK_X_FOUND.trans.x - NOZZLE_RADIUS) + STICK_OUT;
    WaitTime\InPos, 0.5;

ENDIF
    WaitTime\InPos, 0.5;
   I_LOVE_ROBOTS:
    ENDPROC

